(* IEC 61131-3 sources: B-R/Processes/EDT (part 4) *)

(* ---- EDTP4S1C_ACTION.st ---- *)
ACTION P4S1C_ACT:
	//设定时间
	FOR i := 0 TO EDTP4S1_STEP_NUM DO
		IF EDTP4S1C_ST[i] < T#5s THEN
			EDTP4S1C_ST[i] := T#5s;
		END_IF;
		EDTP4S1C_STEP[i].set_time := EDTP4S1C_ST[i];
	END_FOR;

	//流程步骤
	ProcessHandleFC(EDTP4S1C,EDTP4S1C_STEP[0],EDTP4S1_STEP_NUM);

	//object 手自动切换
	IF (EDTP4S1C.status.mode <> 0) AND (NOT EDTP4S1C.auto_mode_edge) THEN
		EDTP4S1C.auto_mode_edge := TRUE;
		EDTP4S1C.manual_mode_edge := FALSE;

		EDTXV1011.control.auto_operate := TRUE;
		EDTXV1022.control.auto_operate := TRUE;
		EDTP16.control.auto_operate := TRUE;
		EDTLV1002.control.auto_operate := TRUE;
		STFP06.control.auto_operate := TRUE;
		STFLV0602.control.auto_operate := TRUE;
		STFLV0601.control.auto_operate := TRUE;
		EDTLV1003.control.auto_operate := TRUE;
		EDTFQV1001C.control.auto_operate := TRUE;
		EDTTV1006B.control.auto_operate := TRUE;
		EDTXV1023.control.auto_operate := TRUE;
		EDTXV1018.control.auto_operate := TRUE;
		EDTTV1005A.control.auto_operate := TRUE;
		EDTTV1005B.control.auto_operate := TRUE;
		EDTTV1006A.control.auto_operate := TRUE;
		EDTXV1020.control.auto_operate := TRUE;
		EDTR04C.control.auto_operate := TRUE;
		EDTLV1004C.control.auto_operate := TRUE;
	END_IF;

	IF (EDTP4S1C.status.mode = 0) AND (NOT EDTP4S1C.manual_mode_edge) THEN
		EDTP4S1C.manual_mode_edge := TRUE;
		EDTP4S1C.auto_mode_edge := FALSE;

		EDTXV1011.control.manual_operate := TRUE;
		EDTXV1022.control.manual_operate := TRUE;
		EDTP16.control.manual_operate := TRUE;
		EDTLV1002.control.manual_operate := TRUE;
		STFP06.control.manual_operate := TRUE;
		STFLV0602.control.manual_operate := TRUE;
		STFLV0601.control.manual_operate := TRUE;
		EDTLV1003.control.manual_operate := TRUE;
		EDTFQV1001C.control.manual_operate := TRUE;
		EDTTV1006B.control.manual_operate := TRUE;
		EDTXV1023.control.manual_operate := TRUE;
		EDTXV1018.control.manual_operate := TRUE;
		EDTTV1005A.control.manual_operate := TRUE;
		EDTTV1005B.control.manual_operate := TRUE;
		EDTTV1006A.control.manual_operate := TRUE;
		EDTXV1020.control.manual_operate := TRUE;
		EDTR04C.control.manual_operate := TRUE;
		EDTLV1004C.control.manual_operate := TRUE;
	END_IF;

	//错误信号停机
	EDTP4S1C.input.error_signal := (EDTXV1011.status.valve_status >= 2) OR
	(EDTXV1022.status.valve_status >= 2) OR (EDTP16.status.motor_status >= 2) OR
	(EDTLV1002.status.valve_status >= 2) OR (STFP06.status.motor_status >= 2) OR (STFLV0602.status.valve_status >= 2) OR
	(STFLV0601.status.valve_status >= 2) OR (EDTLV1003.status.valve_status >= 2) OR (EDTFQV1001C.status.valve_status >= 2) OR
	(EDTTV1006B.status.valve_status >= 2) OR (EDTXV1023.status.valve_status >= 2) OR
	(EDTXV1018.status.valve_status >= 2) OR (EDTTV1005A.status.valve_status >= 2) OR (EDTTV1005B.status.valve_status >= 2) OR
	(EDTTV1006A.status.valve_status >= 2) OR (EDTR04C.status.motor_status >= 2) OR (EDTXV1020.status.valve_status >= 2);

	//EDTLV1004C自动补水
	//	IF EDTTIT1005.status.value >= EDTP4S1C_PARA_Temp7 THEN
	//		EDTLV1004C.input.auto_open_signal := TRUE;
	//	ELSIF EDTTIT1005.status.value <= (EDTP4S1C_PARA_Temp7 - EDTP4S1C_PARA_Temp8) THEN
	//		EDTLV1004C.input.auto_open_signal := FALSE;
	//	END_IF;
	IF r04c_water THEN
		CASE r04c_water_step OF
			0:
				EDTLV1004C.control.auto_operate := TRUE;
				r04c_water_step := 1;
			1:
				EDTLV1004C.input.auto_open_signal := TRUE;
				r04c_temp := EDTTIT1005.status.value;
				r04c_water_step := 2;
			2:
				IF r04c_temp - EDTTIT1005.status.value >= EDTP4S1C_PARA_Temp8 THEN
					EDTLV1004C.input.auto_open_signal := FALSE;
					r04c_water_step := 0;
					r04c_water := FALSE;
				END_IF;
		END_CASE;
	END_IF;

	IF EDTP4S1C.status.run_state = 1 THEN
		CASE EDTP4S1C.status.run_step OF
			0:
				IF NOT EDTP4S1C_STEP[0].done THEN
					EDTXV1011.control.auto_operate := TRUE;
					EDTXV1022.control.auto_operate := TRUE;
					EDTP16.control.auto_operate := TRUE;
					EDTLV1002.control.auto_operate := TRUE;
					STFP06.control.auto_operate := TRUE;
					STFLV0602.control.auto_operate := TRUE;
					STFLV0601.control.auto_operate := TRUE;
					EDTLV1003.control.auto_operate := TRUE;
					EDTFQV1001C.control.auto_operate := TRUE;
					EDTTV1006B.control.auto_operate := TRUE;
					EDTXV1023.control.auto_operate := TRUE;
					EDTXV1018.control.auto_operate := TRUE;
					EDTTV1005A.control.auto_operate := TRUE;
					EDTTV1005B.control.auto_operate := TRUE;
					EDTTV1006A.control.auto_operate := TRUE;
					EDTXV1020.control.auto_operate := TRUE;
					EDTR04C.control.auto_operate := TRUE;
					EDTLV1004C.control.auto_operate := TRUE;
					EDTP4S1C_STEP[0].done := TRUE;
				END_IF;
			1:
				//手动进DMSO和纯水
			2:
				EDTTV1005A.input.auto_open_signal := TRUE;
				EDTTV1005B.input.auto_open_signal := TRUE;
				EDTXV1023.input.auto_open_signal := TRUE;
				EDTXV1018.input.auto_open_signal := TRUE;
				EDTR04C.input.auto_run_signal := TRUE;
				EDTTV1006B.input.auto_open_signal := TRUE;
				EDTXV1020.input.auto_open_signal := TRUE;
				IF EDTXV1023.input.open_feedback_state AND EDTXV1018.input.open_feedback_state AND EDTR04C.input.run_feedback
					AND EDTTV1006B.input.open_feedback_state AND EDTXV1020.input.open_feedback_state THEN
					EDTP4S1C_STEP[2].done := TRUE;
				END_IF;
			3:
				CASE p4_step1_3c OF
					0:
						IF NOT EDTP4S1C_STEP[3].done THEN
							p4_step1_3c := 1;
						END_IF;
					1:
						R04C_heat := TRUE;
						p4_step1_3c := 2;
					2:
						IF EDTTIT1005.status.value >= EDTP4S1C_PARA_Temp1 THEN
							EDTTV1006B.input.auto_open_signal := FALSE;
							IF EDTTV1006B.input.close_feedback_state THEN
								EDTTV1006A.input.auto_open_signal := TRUE;
								IF EDTTV1006A.input.open_feedback_state THEN
									p4_step1_3c := 3;
								END_IF;
							END_IF;
						END_IF;
					3:
						TON_77.PT := DINT_TO_TIME(EDTP4S1C_PARA_T4 * 3600 * 1000);
						IF EDTTIT1005.status.value >= EDTP4S1C_PARA_Temp2 THEN
							R04C_heat := FALSE;
							R04C_hold := TRUE;
							TON_77.IN := TRUE;
						END_IF;
						IF TON_77.Q THEN
							TON_77.IN := FALSE;
							p4_step1_3c := 4;
						END_IF;
					4:
						p4_step1_3c := 0;
						EDTP4S1C_STEP[3].done := TRUE;
				END_CASE;
				TON_77();
			4:
				//人工取样,确认反应结束
			5:
				R04C_hold := FALSE;
				EDTTV1005A.input.auto_open_signal := FALSE;
				EDTTV1005B.input.auto_open_signal := FALSE;
				IF EDTTV1005A.input.close_feedback_state AND EDTTV1005B.input.close_feedback_state THEN
					EDTP4S1C_STEP[5].done := TRUE;
				END_IF;
			6:
				IF EDTTIT1005.status.value <= EDTP4S1C_PARA_Temp5 THEN
					//					EDTXV1023.input.auto_open_signal := FALSE;
					//					EDTXV1018.input.auto_open_signal := FALSE;
					EDTTV1006A.input.auto_open_signal := FALSE;
				END_IF;
				IF (*EDTXV1023.input.close_feedback_state AND EDTXV1018.input.close_feedback_state AND *)(NOT EDTR04C.input.run_feedback)
					AND EDTTV1006A.input.close_feedback_state THEN
					EDTP4S1C_STEP[6].done := TRUE;
				END_IF;
			7:
				//转移
			8:
				EDTR04C.input.auto_run_signal := FALSE;
				IF NOT EDTR04C.input.run_feedback THEN
					EDTP4S1C_STEP[8].done := TRUE;
				END_IF;
		END_CASE;
	END_IF;

	Slope_2(value := EDTTIT1005.status.value, sample_time := EDTP4S1C_PARA_T5);

	IF R04C_heat THEN
		IF Slope_2.out <= EDTP4S1C_PARA_Slope1 THEN
			EDTTV1005A.input.auto_open_signal := TRUE;
			EDTTV1005B.input.auto_open_signal := TRUE;
		END_IF;
		IF Slope_2.out > EDTP4S1C_PARA_Slope1 AND Slope_2.out <= EDTP4S1C_PARA_Slope2 THEN
			EDTTV1005A.input.auto_open_signal := TRUE;
			EDTTV1005B.input.auto_open_signal := FALSE;
		END_IF;
		IF Slope_2.out > EDTP4S1C_PARA_Slope2 AND Slope_2.out <= EDTP4S1C_PARA_Slope3 THEN
			EDTTV1005A.input.auto_open_signal := FALSE;
			EDTTV1005B.input.auto_open_signal := TRUE;
		END_IF;
		IF Slope_2.out > EDTP4S1C_PARA_Slope3 THEN
			EDTTV1005A.input.auto_open_signal := FALSE;
			EDTTV1005B.input.auto_open_signal := FALSE;
		END_IF;
	END_IF;

	//155-158 大  158-162小阀 162都关
	IF R04C_hold THEN
		IF EDTTIT1005.status.value < EDTP4S1C_PARA_Temp2 THEN
			EDTTV1005A.input.auto_open_signal := TRUE;
			EDTTV1005B.input.auto_open_signal := TRUE;
		END_IF;
		IF EDTTIT1005.status.value < EDTP4S1C_PARA_Temp3 AND EDTTIT1005.status.value >= (EDTP4S1C_PARA_Temp2 + EDTP4S1C_PARA_Temp6) THEN
			EDTTV1005A.input.auto_open_signal := TRUE;
			EDTTV1005B.input.auto_open_signal := FALSE;
		END_IF;
		IF EDTTIT1005.status.value < EDTP4S1C_PARA_Temp4 AND EDTTIT1005.status.value >= (EDTP4S1C_PARA_Temp3 + EDTP4S1C_PARA_Temp6) THEN
			EDTTV1005A.input.auto_open_signal := FALSE;
			EDTTV1005B.input.auto_open_signal := TRUE;
		END_IF;
		IF EDTTIT1005.status.value >= (EDTP4S1C_PARA_Temp4 + EDTP4S1C_PARA_Temp6) THEN
			EDTTV1005A.input.auto_open_signal := FALSE;
			EDTTV1005B.input.auto_open_signal := FALSE;
		END_IF;
	END_IF;

	//======================================================================================================
	//DMSO进料
	//从罐区进料
	IF pot_to_r04_c THEN
		CASE pot_to_r04_c_step OF
			0:
				EDTFQV1001C.input.auto_open_signal := TRUE;
				EDTLV1003.input.auto_open_signal := TRUE;
				STFLV0601.input.auto_open_signal := FALSE;
				STFLV0602.input.auto_open_signal := FALSE;
				IF EDTFQV1001C.input.open_feedback_state AND EDTLV1003.input.open_feedback_state AND
					STFLV0601.input.close_feedback_state AND STFLV0602.input.close_feedback_state THEN
					pot_to_r04_c_step := 1;
				END_IF;
			1:
				LiquidTransfer_30(sp_time := DINT_TO_TIME(EDTP4S1C_PARA_T2 * 1000),
				sp_accumulation := EDTP4S1C_PARA_AC1,
				done := pot_to_r04_c_step_1_done,
				flowmeter := EDTFQIT1001);
				STFP06.input.auto_run_signal := LiquidTransfer_30.run;
				IF pot_to_r04_c_step_1_done AND (NOT STFP06.input.run_feedback) AND (NOT STFP06.input.auto_run_signal) THEN
					pot_to_r04_c_step_1_done := FALSE;
					pot_to_r04_c_step := 2;
				END_IF;
			2:
				IF EDTFQIT1001.flowrate <= flowrate_threshold THEN
					pot_to_r04_c_step := 3;
				END_IF;
			3:
				EDTFQV1001C.input.auto_open_signal := FALSE;
				EDTLV1003.input.auto_open_signal := FALSE;
				IF EDTFQV1001C.input.close_feedback_state AND EDTLV1003.input.close_feedback_state THEN
					pot_to_r04_c_step := 0;
					pot_to_r04_c := FALSE;
				END_IF;
		END_CASE;
	END_IF;

	//从V52进料
	IF v52_to_r04_c THEN
		CASE v52_to_r04_c_step OF
			0:
				EDTFQV1001C.input.auto_open_signal := TRUE;
				EDTLV1002.input.auto_open_signal := TRUE;
				IF EDTFQV1001C.input.open_feedback_state AND EDTLV1002.input.open_feedback_state THEN
					v52_to_r04_c_step := 1;
				END_IF;
			1:
				LiquidTransfer_31(sp_time := DINT_TO_TIME(EDTP4S1C_PARA_T3 * 1000),
				sp_accumulation := EDTP4S1C_PARA_AC2,
				done := v52_to_r04_c_step_1_done,
				flowmeter := EDTFQIT1001);
				EDTP16.input.auto_run_signal := LiquidTransfer_31.run;
				IF v52_to_r04_c_step_1_done AND (NOT EDTP16.input.run_feedback) AND (NOT EDTP16.input.auto_run_signal) THEN
					v52_to_r04_c_step_1_done := FALSE;
					v52_to_r04_c_step := 2;
				END_IF;
			2:
				IF EDTFQIT1001.flowrate <= flowrate_threshold THEN
					v52_to_r04_c_step := 3;
				END_IF;
			3:
				EDTFQV1001C.input.auto_open_signal := FALSE;
				EDTLV1002.input.auto_open_signal := FALSE;
				IF EDTFQV1001C.input.close_feedback_state AND EDTLV1002.input.close_feedback_state THEN
					v52_to_r04_c_step := 0;
					v52_to_r04_c := FALSE;
				END_IF;
		END_CASE;
	END_IF;

	//=======================================================================================================
	//人工确认步骤可用
	IF (EDTP4S1C.status.run_state) AND (NOT EDTP4S1C_STEP[EDTP4S1C.status.run_step].done AND ((EDTP4S1C.status.run_step = 1) OR (EDTP4S1C.status.run_step = 4) OR (EDTP4S1C.status.run_step = 7))) THEN
		EDTP4S1C.status.confirm_enable := TRUE;
	ELSE
		EDTP4S1C.status.confirm_enable := FALSE;
	END_IF;
END_ACTION

(* ---- EDTP4S1D_ACTION.st ---- *)
ACTION P4S1D_ACT:
	//设定时间
	FOR i := 0 TO EDTP4S1_STEP_NUM DO
		IF EDTP4S1D_ST[i] < T#5s THEN
			EDTP4S1D_ST[i] := T#5s;
		END_IF;
		EDTP4S1D_STEP[i].set_time := EDTP4S1D_ST[i];
	END_FOR;

	//流程步骤
	ProcessHandleFC(EDTP4S1D,EDTP4S1D_STEP[0],EDTP4S1_STEP_NUM);

	//object 手自动切换
	IF (EDTP4S1D.status.mode <> 0) AND (NOT EDTP4S1D.auto_mode_edge) THEN
		EDTP4S1D.auto_mode_edge := TRUE;
		EDTP4S1D.manual_mode_edge := FALSE;

		EDTXV1011.control.auto_operate := TRUE;
		EDTXV1022.control.auto_operate := TRUE;
		EDTP16.control.auto_operate := TRUE;
		EDTLV1002.control.auto_operate := TRUE;
		STFP06.control.auto_operate := TRUE;
		STFLV0602.control.auto_operate := TRUE;
		STFLV0601.control.auto_operate := TRUE;
		EDTLV1003.control.auto_operate := TRUE;
		EDTFQV1001D.control.auto_operate := TRUE;
		EDTTV1008B.control.auto_operate := TRUE;
		EDTXV1024.control.auto_operate := TRUE;
		EDTXV1019.control.auto_operate := TRUE;
		EDTTV1007A.control.auto_operate := TRUE;
		EDTTV1007B.control.auto_operate := TRUE;
		EDTTV1008A.control.auto_operate := TRUE;
		EDTXV1021.control.auto_operate := TRUE;
		EDTR04D.control.auto_operate := TRUE;
		EDTLV1004D.control.auto_operate := TRUE;
	END_IF;

	IF (EDTP4S1D.status.mode = 0) AND (NOT EDTP4S1D.manual_mode_edge) THEN
		EDTP4S1D.manual_mode_edge := TRUE;
		EDTP4S1D.auto_mode_edge := FALSE;

		EDTXV1011.control.manual_operate := TRUE;
		EDTXV1022.control.manual_operate := TRUE;
		EDTP16.control.manual_operate := TRUE;
		EDTLV1002.control.manual_operate := TRUE;
		STFP06.control.manual_operate := TRUE;
		STFLV0602.control.manual_operate := TRUE;
		STFLV0601.control.manual_operate := TRUE;
		EDTLV1003.control.manual_operate := TRUE;
		EDTFQV1001D.control.manual_operate := TRUE;
		EDTTV1008B.control.manual_operate := TRUE;
		EDTXV1024.control.manual_operate := TRUE;
		EDTXV1019.control.manual_operate := TRUE;
		EDTTV1007A.control.manual_operate := TRUE;
		EDTTV1007B.control.manual_operate := TRUE;
		EDTTV1008A.control.manual_operate := TRUE;
		EDTXV1021.control.manual_operate := TRUE;
		EDTR04D.control.manual_operate := TRUE;
		EDTLV1004D.control.manual_operate := TRUE;
	END_IF;

	//错误信号停机
	EDTP4S1D.input.error_signal := (EDTXV1011.status.valve_status >= 2) OR
	(EDTXV1022.status.valve_status >= 2) OR (EDTP16.status.motor_status >= 2) OR
	(EDTLV1002.status.valve_status >= 2) OR (STFP06.status.motor_status >= 2) OR (STFLV0602.status.valve_status >= 2) OR
	(STFLV0601.status.valve_status >= 2) OR (EDTLV1003.status.valve_status >= 2) OR (EDTFQV1001D.status.valve_status >= 2) OR
	(EDTTV1008B.status.valve_status >= 2) OR (EDTXV1024.status.valve_status >= 2) OR
	(EDTXV1019.status.valve_status >= 2) OR (EDTTV1007A.status.valve_status >= 2) OR (EDTTV1007B.status.valve_status >= 2) OR
	(EDTTV1008A.status.valve_status >= 2) OR (EDTR04D.status.motor_status >= 2) OR (EDTXV1021.status.valve_status >= 2);

	//EDTLV1004D自动补水
	//	IF EDTTIT1007.status.value >= EDTP4S1D_PARA_Temp7 THEN
	//		EDTLV1004D.input.auto_open_signal := TRUE;
	//	ELSIF EDTTIT1007.status.value <= (EDTP4S1D_PARA_Temp7 - EDTP4S1D_PARA_Temp8) THEN
	//		EDTLV1004D.input.auto_open_signal := FALSE;
	//	END_IF;
	IF r04d_water THEN
		CASE r04d_water_step OF
			0:
				EDTLV1004D.control.auto_operate := TRUE;
				r04d_water_step := 1;
			1:
				EDTLV1004D.input.auto_open_signal := TRUE;
				r04d_temp := EDTTIT1007.status.value;
				r04d_water_step := 2;
			2:
				IF r04d_temp - EDTTIT1007.status.value >= EDTP4S1D_PARA_Temp8 THEN
					EDTLV1004D.input.auto_open_signal := FALSE;
					r04d_water_step := 0;
					r04d_water := FALSE;
				END_IF;
		END_CASE;
	END_IF;

	IF EDTP4S1D.status.run_state = 1 THEN
		CASE EDTP4S1D.status.run_step OF
			0:
				IF NOT EDTP4S1D_STEP[0].done THEN
					EDTXV1011.control.auto_operate := TRUE;
					EDTXV1022.control.auto_operate := TRUE;
					EDTP16.control.auto_operate := TRUE;
					EDTLV1002.control.auto_operate := TRUE;
					STFP06.control.auto_operate := TRUE;
					STFLV0602.control.auto_operate := TRUE;
					STFLV0601.control.auto_operate := TRUE;
					EDTLV1003.control.auto_operate := TRUE;
					EDTFQV1001D.control.auto_operate := TRUE;
					EDTTV1008B.control.auto_operate := TRUE;
					EDTXV1024.control.auto_operate := TRUE;
					EDTXV1019.control.auto_operate := TRUE;
					EDTTV1007A.control.auto_operate := TRUE;
					EDTTV1007B.control.auto_operate := TRUE;
					EDTTV1008A.control.auto_operate := TRUE;
					EDTXV1021.control.auto_operate := TRUE;
					EDTR04D.control.auto_operate := TRUE;
					EDTLV1004D.control.auto_operate := TRUE;
					EDTP4S1D_STEP[0].done := TRUE;
				END_IF;
			1:
				//手动进DMSO和纯水
			2:
				EDTTV1007A.input.auto_open_signal := TRUE;
				EDTTV1007B.input.auto_open_signal := TRUE;
				EDTXV1024.input.auto_open_signal := TRUE;
				EDTXV1019.input.auto_open_signal := TRUE;
				EDTR04D.input.auto_run_signal := TRUE;
				EDTTV1008B.input.auto_open_signal := TRUE;
				EDTXV1021.input.auto_open_signal := TRUE;
				IF EDTXV1024.input.open_feedback_state AND EDTXV1019.input.open_feedback_state AND EDTR04D.input.run_feedback
					AND EDTTV1008B.input.open_feedback_state AND EDTXV1021.input.open_feedback_state THEN
					EDTP4S1D_STEP[2].done := TRUE;
				END_IF;
			3:
				CASE p4_step1_3d OF
					0:
						IF NOT EDTP4S1D_STEP[3].done THEN
							p4_step1_3d := 1;
						END_IF;
					1:
						R04D_heat := TRUE;
						p4_step1_3d := 2;
					2:
						IF EDTTIT1007.status.value >= EDTP4S1D_PARA_Temp1 THEN
							EDTTV1008B.input.auto_open_signal := FALSE;
							IF EDTTV1008B.input.close_feedback_state THEN
								EDTTV1008A.input.auto_open_signal := TRUE;
								IF EDTTV1008A.input.open_feedback_state THEN
									p4_step1_3d := 3;
								END_IF;
							END_IF;
						END_IF;
					3:
						TON_79.PT := DINT_TO_TIME(EDTP4S1D_PARA_T4 * 3600 * 1000);
						IF EDTTIT1007.status.value >= EDTP4S1D_PARA_Temp2 THEN
							R04D_heat := FALSE;
							R04D_hold := TRUE;
							TON_79.IN := TRUE;
						END_IF;
						IF TON_79.Q THEN
							TON_79.IN := FALSE;
							p4_step1_3d := 4;
						END_IF;
					4:
						p4_step1_3d := 0;
						EDTP4S1D_STEP[3].done := TRUE;
				END_CASE;
				TON_79();
			4:
				//人工取样,确认反应结束
			5:
				R04D_hold := FALSE;
				EDTTV1007A.input.auto_open_signal := FALSE;
				EDTTV1007B.input.auto_open_signal := FALSE;
				IF EDTTV1007A.input.close_feedback_state AND EDTTV1007B.input.close_feedback_state THEN
					EDTP4S1D_STEP[5].done := TRUE;
				END_IF;
			6:
				IF EDTTIT1007.status.value <= EDTP4S1D_PARA_Temp5 THEN
					//					EDTXV1024.input.auto_open_signal := FALSE;
					//					EDTXV1019.input.auto_open_signal := FALSE;
					EDTTV1008A.input.auto_open_signal := FALSE;
				END_IF;
				IF (*EDTXV1024.input.close_feedback_state AND EDTXV1019.input.close_feedback_state AND *)(NOT EDTR04D.input.run_feedback)
					AND EDTTV1008A.input.close_feedback_state THEN
					EDTP4S1D_STEP[6].done := TRUE;
				END_IF;
			7:
				//转移
			8:
				EDTR04D.input.auto_run_signal := FALSE;
				IF NOT EDTR04D.input.run_feedback THEN
					EDTP4S1D_STEP[8].done := TRUE;
				END_IF;
		END_CASE;
	END_IF;

	Slope_3(value := EDTTIT1007.status.value, sample_time := EDTP4S1D_PARA_T5);

	IF R04D_heat THEN
		IF Slope_3.out <= EDTP4S1D_PARA_Slope1 THEN
			EDTTV1007A.input.auto_open_signal := TRUE;
			EDTTV1007B.input.auto_open_signal := TRUE;
		END_IF;
		IF Slope_3.out > EDTP4S1D_PARA_Slope1 AND Slope_3.out <= EDTP4S1D_PARA_Slope2 THEN
			EDTTV1007A.input.auto_open_signal := TRUE;
			EDTTV1007B.input.auto_open_signal := FALSE;
		END_IF;
		IF Slope_3.out > EDTP4S1D_PARA_Slope2 AND Slope_3.out <= EDTP4S1D_PARA_Slope3 THEN
			EDTTV1007A.input.auto_open_signal := FALSE;
			EDTTV1007B.input.auto_open_signal := TRUE;
		END_IF;
		IF Slope_3.out > EDTP4S1D_PARA_Slope3 THEN
			EDTTV1007A.input.auto_open_signal := FALSE;
			EDTTV1007B.input.auto_open_signal := FALSE;
		END_IF;
	END_IF;

	//155-158 大  158-162小阀 162都关
	IF R04D_hold THEN
		IF EDTTIT1007.status.value < EDTP4S1D_PARA_Temp2 THEN
			EDTTV1007A.input.auto_open_signal := TRUE;
			EDTTV1007B.input.auto_open_signal := TRUE;
		END_IF;
		IF EDTTIT1007.status.value < EDTP4S1D_PARA_Temp3 AND EDTTIT1007.status.value >= (EDTP4S1D_PARA_Temp2 + EDTP4S1D_PARA_Temp6) THEN
			EDTTV1007A.input.auto_open_signal := TRUE;
			EDTTV1007B.input.auto_open_signal := FALSE;
		END_IF;
		IF EDTTIT1007.status.value < EDTP4S1D_PARA_Temp4 AND EDTTIT1007.status.value >= (EDTP4S1D_PARA_Temp3 + EDTP4S1D_PARA_Temp6) THEN
			EDTTV1007A.input.auto_open_signal := FALSE;
			EDTTV1007B.input.auto_open_signal := TRUE;
		END_IF;
		IF EDTTIT1007.status.value >= (EDTP4S1D_PARA_Temp4 + EDTP4S1D_PARA_Temp6) THEN
			EDTTV1007A.input.auto_open_signal := FALSE;
			EDTTV1007B.input.auto_open_signal := FALSE;
		END_IF;
	END_IF;

	//======================================================================================================
	//DMSO进料
	//从罐区进料
	IF pot_to_r04_d THEN
		CASE pot_to_r04_d_step OF
			0:
				EDTFQV1001D.input.auto_open_signal := TRUE;
				EDTLV1003.input.auto_open_signal := TRUE;
				STFLV0601.input.auto_open_signal := FALSE;
				STFLV0602.input.auto_open_signal := FALSE;
				IF EDTFQV1001D.input.open_feedback_state AND EDTLV1003.input.open_feedback_state AND
					STFLV0601.input.close_feedback_state AND STFLV0602.input.close_feedback_state THEN
					pot_to_r04_d_step := 1;
				END_IF;
			1:
				LiquidTransfer_32(sp_time := DINT_TO_TIME(EDTP4S1D_PARA_T2 * 1000),
				sp_accumulation := EDTP4S1D_PARA_AC1,
				done := pot_to_r04_d_step_1_done,
				flowmeter := EDTFQIT1001);
				STFP06.input.auto_run_signal := LiquidTransfer_32.run;
				IF pot_to_r04_d_step_1_done AND (NOT STFP06.input.run_feedback) AND (NOT STFP06.input.auto_run_signal) THEN
					pot_to_r04_d_step_1_done := FALSE;
					pot_to_r04_d_step := 2;
				END_IF;
			2:
				IF EDTFQIT1001.flowrate <= flowrate_threshold THEN
					pot_to_r04_d_step := 3;
				END_IF;
			3:
				EDTFQV1001D.input.auto_open_signal := FALSE;
				EDTLV1003.input.auto_open_signal := FALSE;
				IF EDTFQV1001D.input.close_feedback_state AND EDTLV1003.input.close_feedback_state THEN
					pot_to_r04_d_step := 0;
					pot_to_r04_d := FALSE;
				END_IF;
		END_CASE;
	END_IF;

	//从V52进料
	IF v52_to_r04_d THEN
		CASE v52_to_r04_d_step OF
			0:
				EDTFQV1001D.input.auto_open_signal := TRUE;
				EDTLV1002.input.auto_open_signal := TRUE;
				IF EDTFQV1001D.input.open_feedback_state AND EDTLV1002.input.open_feedback_state THEN
					v52_to_r04_d_step := 1;
				END_IF;
			1:
				LiquidTransfer_33(sp_time := DINT_TO_TIME(EDTP4S1D_PARA_T3 * 1000),
				sp_accumulation := EDTP4S1D_PARA_AC2,
				done := v52_to_r04_d_step_1_done,
				flowmeter := EDTFQIT1001);
				EDTP16.input.auto_run_signal := LiquidTransfer_33.run;
				IF v52_to_r04_d_step_1_done AND (NOT EDTP16.input.run_feedback) AND (NOT EDTP16.input.auto_run_signal) THEN
					v52_to_r04_d_step_1_done := FALSE;
					v52_to_r04_d_step := 2;
				END_IF;
			2:
				IF EDTFQIT1001.flowrate <= flowrate_threshold THEN
					v52_to_r04_d_step := 3;
				END_IF;
			3:
				EDTFQV1001D.input.auto_open_signal := FALSE;
				EDTLV1002.input.auto_open_signal := FALSE;
				IF EDTFQV1001D.input.close_feedback_state AND EDTLV1002.input.close_feedback_state THEN
					v52_to_r04_d_step := 0;
					v52_to_r04_d := FALSE;
				END_IF;
		END_CASE;
	END_IF;

	//=======================================================================================================
	//人工确认步骤可用
	IF (EDTP4S1D.status.run_state) AND (NOT EDTP4S1D_STEP[EDTP4S1D.status.run_step].done AND ((EDTP4S1D.status.run_step = 1) OR (EDTP4S1D.status.run_step = 4) OR (EDTP4S1D.status.run_step = 7))) THEN
		EDTP4S1D.status.confirm_enable := TRUE;
	ELSE
		EDTP4S1D.status.confirm_enable := FALSE;
	END_IF;
END_ACTION

(* ---- EDTP4S1E_ACTION.st ---- *)
ACTION P4S1E_ACT:
	//设定时间
	FOR i := 0 TO EDTP4S1_STEP_NUM DO
		IF EDTP4S1E_ST[i] < T#5s THEN
			EDTP4S1E_ST[i] := T#5s;
		END_IF;
		EDTP4S1E_STEP[i].set_time := EDTP4S1E_ST[i];
	END_FOR;

	//流程步骤
	ProcessHandleFC(EDTP4S1E,EDTP4S1E_STEP[0],EDTP4S1_STEP_NUM);

	//object 手自动切换
	IF (EDTP4S1E.status.mode <> 0) AND (NOT EDTP4S1E.auto_mode_edge) THEN
		EDTP4S1E.auto_mode_edge := TRUE;
		EDTP4S1E.manual_mode_edge := FALSE;

		EDTXV1011.control.auto_operate := TRUE;
		EDTXV1031.control.auto_operate := TRUE;
		EDTP16.control.auto_operate := TRUE;
		EDTLV1002.control.auto_operate := TRUE;
		STFP06.control.auto_operate := TRUE;
		STFLV0602.control.auto_operate := TRUE;
		STFLV0601.control.auto_operate := TRUE;
		EDTLV1003.control.auto_operate := TRUE;
		EDTFQV1001E.control.auto_operate := TRUE;
		EDTTV1010B.control.auto_operate := TRUE;
		EDTXV1032.control.auto_operate := TRUE;
		EDTXV1027.control.auto_operate := TRUE;
		EDTTV1009A.control.auto_operate := TRUE;
		EDTTV1009B.control.auto_operate := TRUE;
		EDTTV1010A.control.auto_operate := TRUE;
		EDTXV1029.control.auto_operate := TRUE;
		EDTR04E.control.auto_operate := TRUE;
		EDTLV1004E.control.auto_operate := TRUE;
	END_IF;

	IF (EDTP4S1E.status.mode = 0) AND (NOT EDTP4S1E.manual_mode_edge) THEN
		EDTP4S1E.manual_mode_edge := TRUE;
		EDTP4S1E.auto_mode_edge := FALSE;

		EDTXV1011.control.manual_operate := TRUE;
		EDTXV1031.control.manual_operate := TRUE;
		EDTP16.control.manual_operate := TRUE;
		EDTLV1002.control.manual_operate := TRUE;
		STFP06.control.manual_operate := TRUE;
		STFLV0602.control.manual_operate := TRUE;
		STFLV0601.control.manual_operate := TRUE;
		EDTLV1003.control.manual_operate := TRUE;
		EDTFQV1001E.control.manual_operate := TRUE;
		EDTTV1010B.control.manual_operate := TRUE;
		EDTXV1032.control.manual_operate := TRUE;
		EDTXV1027.control.manual_operate := TRUE;
		EDTTV1009A.control.manual_operate := TRUE;
		EDTTV1009B.control.manual_operate := TRUE;
		EDTTV1010A.control.manual_operate := TRUE;
		EDTXV1029.control.manual_operate := TRUE;
		EDTR04E.control.manual_operate := TRUE;
		EDTLV1004E.control.manual_operate := TRUE;
	END_IF;

	//错误信号停机
	EDTP4S1E.input.error_signal := (EDTXV1011.status.valve_status >= 2) OR
	(EDTXV1031.status.valve_status >= 2) OR (EDTP16.status.motor_status >= 2) OR
	(EDTLV1002.status.valve_status >= 2) OR (STFP06.status.motor_status >= 2) OR (STFLV0602.status.valve_status >= 2) OR
	(STFLV0601.status.valve_status >= 2) OR (EDTLV1003.status.valve_status >= 2) OR (EDTFQV1001E.status.valve_status >= 2) OR
	(EDTTV1010B.status.valve_status >= 2) OR (EDTXV1032.status.valve_status >= 2) OR
	(EDTXV1027.status.valve_status >= 2) OR (EDTTV1009A.status.valve_status >= 2) OR (EDTTV1009B.status.valve_status >= 2) OR
	(EDTTV1010A.status.valve_status >= 2) OR (EDTR04E.status.motor_status >= 2) OR (EDTXV1029.status.valve_status >= 2);

	//EDTLV1004E自动补水
	//	IF EDTTIT1009.status.value >= EDTP4S1E_PARA_Temp7 THEN
	//		EDTLV1004E.input.auto_open_signal := TRUE;
	//	ELSIF EDTTIT1009.status.value <= (EDTP4S1E_PARA_Temp7 - EDTP4S1E_PARA_Temp8) THEN
	//		EDTLV1004E.input.auto_open_signal := FALSE;
	//	END_IF;
	IF r04e_water THEN
		CASE r04e_water_step OF
			0:
				EDTLV1004E.control.auto_operate := TRUE;
				r04e_water_step := 1;
			1:
				EDTLV1004E.input.auto_open_signal := TRUE;
				r04e_temp := EDTTIT1009.status.value;
				r04e_water_step := 2;
			2:
				IF r04e_temp - EDTTIT1009.status.value >= EDTP4S1E_PARA_Temp8 THEN
					EDTLV1004E.input.auto_open_signal := FALSE;
					r04e_water_step := 0;
					r04e_water := FALSE;
				END_IF;
		END_CASE;
	END_IF;

	IF EDTP4S1E.status.run_state = 1 THEN
		CASE EDTP4S1E.status.run_step OF
			0:
				IF NOT EDTP4S1E_STEP[0].done THEN
					EDTXV1011.control.auto_operate := TRUE;
					EDTXV1031.control.auto_operate := TRUE;
					EDTP16.control.auto_operate := TRUE;
					EDTLV1002.control.auto_operate := TRUE;
					STFP06.control.auto_operate := TRUE;
					STFLV0602.control.auto_operate := TRUE;
					STFLV0601.control.auto_operate := TRUE;
					EDTLV1003.control.auto_operate := TRUE;
					EDTFQV1001E.control.auto_operate := TRUE;
					EDTTV1010B.control.auto_operate := TRUE;
					EDTXV1032.control.auto_operate := TRUE;
					EDTXV1027.control.auto_operate := TRUE;
					EDTTV1009A.control.auto_operate := TRUE;
					EDTTV1009B.control.auto_operate := TRUE;
					EDTTV1010A.control.auto_operate := TRUE;
					EDTXV1029.control.auto_operate := TRUE;
					EDTR04E.control.auto_operate := TRUE;
					EDTLV1004E.control.auto_operate := TRUE;
					EDTP4S1E_STEP[0].done := TRUE;
				END_IF;
			1:
				//手动进DMSO和纯水
			2:
				EDTTV1009A.input.auto_open_signal := TRUE;
				EDTTV1009B.input.auto_open_signal := TRUE;
				EDTXV1032.input.auto_open_signal := TRUE;
				EDTXV1027.input.auto_open_signal := TRUE;
				EDTR04E.input.auto_run_signal := TRUE;
				EDTTV1010B.input.auto_open_signal := TRUE;
				EDTXV1029.input.auto_open_signal := TRUE;
				IF EDTXV1032.input.open_feedback_state AND EDTXV1027.input.open_feedback_state AND EDTR04E.input.run_feedback
					AND EDTTV1010B.input.open_feedback_state AND EDTXV1029.input.open_feedback_state THEN
					EDTP4S1E_STEP[2].done := TRUE;
				END_IF;
			3:
				CASE p4_step1_3e OF
					0:
						IF NOT EDTP4S1E_STEP[3].done THEN
							p4_step1_3e := 1;
						END_IF;
					1:
						R04E_heat := TRUE;
						p4_step1_3e := 2;
					2:
						IF EDTTIT1009.status.value >= EDTP4S1E_PARA_Temp1 THEN
							EDTTV1010B.input.auto_open_signal := FALSE;
							IF EDTTV1010B.input.close_feedback_state THEN
								EDTTV1010A.input.auto_open_signal := TRUE;
								IF EDTTV1010A.input.open_feedback_state THEN
									p4_step1_3e := 3;
								END_IF;
							END_IF;
						END_IF;

					3:
						TON_80.PT := DINT_TO_TIME(EDTP4S1E_PARA_T4 * 3600 * 1000);
						IF EDTTIT1009.status.value >= EDTP4S1E_PARA_Temp2 THEN
							R04E_heat := FALSE;
							R04E_hold := TRUE;
							TON_80.IN := TRUE;
						END_IF;
						IF TON_80.Q THEN
							TON_80.IN := FALSE;
							p4_step1_3e := 4;
						END_IF;
					4:
						p4_step1_3e := 0;
						EDTP4S1E_STEP[3].done := TRUE;
				END_CASE;
				TON_80();
			4:
				//人工取样,确认反应结束
			5:
				R04E_hold := FALSE;
				EDTTV1009A.input.auto_open_signal := FALSE;
				EDTTV1009B.input.auto_open_signal := FALSE;
				IF EDTTV1009A.input.close_feedback_state AND EDTTV1009B.input.close_feedback_state THEN
					EDTP4S1E_STEP[5].done := TRUE;
				END_IF;
			6:
				IF EDTTIT1009.status.value <= EDTP4S1E_PARA_Temp5 THEN
					//					EDTXV1032.input.auto_open_signal := FALSE;
					//					EDTXV1027.input.auto_open_signal := FALSE;
					EDTTV1010A.input.auto_open_signal := FALSE;
				END_IF;
				IF (*EDTXV1032.input.close_feedback_state AND EDTXV1027.input.close_feedback_state AND *)(NOT EDTR04E.input.run_feedback)
					AND EDTTV1010A.input.close_feedback_state THEN
					EDTP4S1E_STEP[6].done := TRUE;
				END_IF;
			7:
				//转移
			8:
				EDTR04E.input.auto_run_signal := FALSE;
				IF NOT EDTR04E.input.run_feedback THEN
					EDTP4S1E_STEP[8].done := TRUE;
				END_IF;
		END_CASE;
	END_IF;

	Slope_4(value := EDTTIT1009.status.value, sample_time := EDTP4S1E_PARA_T5);

	IF R04E_heat THEN
		IF Slope_4.out <= EDTP4S1E_PARA_Slope1 THEN
			EDTTV1009A.input.auto_open_signal := TRUE;
			EDTTV1009B.input.auto_open_signal := TRUE;
		END_IF;
		IF Slope_4.out > EDTP4S1E_PARA_Slope1 AND Slope_4.out <= EDTP4S1E_PARA_Slope2 THEN
			EDTTV1009A.input.auto_open_signal := TRUE;
			EDTTV1009B.input.auto_open_signal := FALSE;
		END_IF;
		IF Slope_4.out > EDTP4S1E_PARA_Slope2 AND Slope_4.out <= EDTP4S1E_PARA_Slope3 THEN
			EDTTV1009A.input.auto_open_signal := FALSE;
			EDTTV1009B.input.auto_open_signal := TRUE;
		END_IF;
		IF Slope_4.out > EDTP4S1E_PARA_Slope3 THEN
			EDTTV1009A.input.auto_open_signal := FALSE;
			EDTTV1009B.input.auto_open_signal := FALSE;
		END_IF;
	END_IF;

	//155-158 大  158-162小阀 162都关
	IF R04E_hold THEN
		IF EDTTIT1009.status.value < EDTP4S1E_PARA_Temp2 THEN
			EDTTV1009A.input.auto_open_signal := TRUE;
			EDTTV1009B.input.auto_open_signal := TRUE;
		END_IF;
		IF EDTTIT1009.status.value < EDTP4S1E_PARA_Temp3 AND EDTTIT1009.status.value >= (EDTP4S1E_PARA_Temp2 + EDTP4S1E_PARA_Temp6) THEN
			EDTTV1009A.input.auto_open_signal := TRUE;
			EDTTV1009B.input.auto_open_signal := FALSE;
		END_IF;
		IF EDTTIT1009.status.value < EDTP4S1E_PARA_Temp4 AND EDTTIT1009.status.value >= (EDTP4S1E_PARA_Temp3 + EDTP4S1E_PARA_Temp6) THEN
			EDTTV1009A.input.auto_open_signal := FALSE;
			EDTTV1009B.input.auto_open_signal := TRUE;
		END_IF;
		IF EDTTIT1009.status.value >= (EDTP4S1E_PARA_Temp4 + EDTP4S1E_PARA_Temp6) THEN
			EDTTV1009A.input.auto_open_signal := FALSE;
			EDTTV1009B.input.auto_open_signal := FALSE;
		END_IF;
	END_IF;

	//======================================================================================================
	//DMSO进料
	//从罐区进料
	IF pot_to_r04_e THEN
		CASE pot_to_r04_e_step OF
			0:
				EDTFQV1001E.input.auto_open_signal := TRUE;
				EDTLV1003.input.auto_open_signal := TRUE;
				STFLV0601.input.auto_open_signal := FALSE;
				STFLV0602.input.auto_open_signal := FALSE;
				IF EDTFQV1001E.input.open_feedback_state AND EDTLV1003.input.open_feedback_state AND
					STFLV0601.input.close_feedback_state AND STFLV0602.input.close_feedback_state THEN
					pot_to_r04_e_step := 1;
				END_IF;
			1:
				LiquidTransfer_34(sp_time := DINT_TO_TIME(EDTP4S1E_PARA_T2 * 1000),
				sp_accumulation := EDTP4S1E_PARA_AC1,
				done := pot_to_r04_e_step_1_done,
				flowmeter := EDTFQIT1001);
				STFP06.input.auto_run_signal := LiquidTransfer_34.run;
				IF pot_to_r04_e_step_1_done AND (NOT STFP06.input.run_feedback) AND (NOT STFP06.input.auto_run_signal) THEN
					pot_to_r04_e_step_1_done := FALSE;
					pot_to_r04_e_step := 2;
				END_IF;
			2:
				IF EDTFQIT1001.flowrate <= flowrate_threshold THEN
					pot_to_r04_e_step := 3;
				END_IF;
			3:
				EDTFQV1001E.input.auto_open_signal := FALSE;
				EDTLV1003.input.auto_open_signal := FALSE;
				IF EDTFQV1001E.input.close_feedback_state AND EDTLV1003.input.close_feedback_state THEN
					pot_to_r04_e_step := 0;
					pot_to_r04_e := FALSE;
				END_IF;
		END_CASE;
	END_IF;

	//从V52进料
	IF v52_to_r04_e THEN
		CASE v52_to_r04_e_step OF
			0:
				EDTFQV1001E.input.auto_open_signal := TRUE;
				EDTLV1002.input.auto_open_signal := TRUE;
				IF EDTFQV1001E.input.open_feedback_state AND EDTLV1002.input.open_feedback_state THEN
					v52_to_r04_e_step := 1;
				END_IF;
			1:
				LiquidTransfer_35(sp_time := DINT_TO_TIME(EDTP4S1E_PARA_T3 * 1000),
				sp_accumulation := EDTP4S1E_PARA_AC2,
				done := v52_to_r04_e_step_1_done,
				flowmeter := EDTFQIT1001);
				EDTP16.input.auto_run_signal := LiquidTransfer_35.run;
				IF v52_to_r04_e_step_1_done AND (NOT EDTP16.input.run_feedback) AND (NOT EDTP16.input.auto_run_signal) THEN
					v52_to_r04_e_step_1_done := FALSE;
					v52_to_r04_e_step := 2;
				END_IF;
			2:
				IF EDTFQIT1001.flowrate <= flowrate_threshold THEN
					v52_to_r04_e_step := 3;
				END_IF;
			3:
				EDTFQV1001E.input.auto_open_signal := FALSE;
				EDTLV1002.input.auto_open_signal := FALSE;
				IF EDTFQV1001E.input.close_feedback_state AND EDTLV1002.input.close_feedback_state THEN
					v52_to_r04_e_step := 0;
					v52_to_r04_e := FALSE;
				END_IF;
		END_CASE;
	END_IF;

	//=======================================================================================================
	//人工确认步骤可用
	IF (EDTP4S1E.status.run_state) AND (NOT EDTP4S1E_STEP[EDTP4S1E.status.run_step].done AND ((EDTP4S1E.status.run_step = 1) OR (EDTP4S1E.status.run_step = 4) OR (EDTP4S1E.status.run_step = 7))) THEN
		EDTP4S1E.status.confirm_enable := TRUE;
	ELSE
		EDTP4S1E.status.confirm_enable := FALSE;
	END_IF;
END_ACTION

(* ---- EDTP4S1F_ACTION.st ---- *)
ACTION P4S1F_ACT:
	//设定时间
	FOR i := 0 TO EDTP4S1_STEP_NUM DO
		IF EDTP4S1F_ST[i] < T#5s THEN
			EDTP4S1F_ST[i] := T#5s;
		END_IF;
		EDTP4S1F_STEP[i].set_time := EDTP4S1F_ST[i];
	END_FOR;

	//流程步骤
	ProcessHandleFC(EDTP4S1F,EDTP4S1F_STEP[0],EDTP4S1_STEP_NUM);

	//object 手自动切换
	IF (EDTP4S1F.status.mode <> 0) AND (NOT EDTP4S1F.auto_mode_edge) THEN
		EDTP4S1F.auto_mode_edge := TRUE;
		EDTP4S1F.manual_mode_edge := FALSE;

		EDTXV1011.control.auto_operate := TRUE;
		EDTXV1031.control.auto_operate := TRUE;
		EDTP16.control.auto_operate := TRUE;
		EDTLV1002.control.auto_operate := TRUE;
		STFP06.control.auto_operate := TRUE;
		STFLV0602.control.auto_operate := TRUE;
		STFLV0601.control.auto_operate := TRUE;
		EDTLV1003.control.auto_operate := TRUE;
		EDTFQV1001F.control.auto_operate := TRUE;
		EDTTV1012B.control.auto_operate := TRUE;
		EDTXV1033.control.auto_operate := TRUE;
		EDTXV1028.control.auto_operate := TRUE;
		EDTTV1011A.control.auto_operate := TRUE;
		EDTTV1011B.control.auto_operate := TRUE;
		EDTTV1012A.control.auto_operate := TRUE;
		EDTXV1030.control.auto_operate := TRUE;
		EDTR04F.control.auto_operate := TRUE;
		EDTLV1004F.control.auto_operate := TRUE;
	END_IF;

	IF (EDTP4S1F.status.mode = 0) AND (NOT EDTP4S1F.manual_mode_edge) THEN
		EDTP4S1F.manual_mode_edge := TRUE;
		EDTP4S1F.auto_mode_edge := FALSE;

		EDTXV1011.control.manual_operate := TRUE;
		EDTXV1031.control.manual_operate := TRUE;
		EDTP16.control.manual_operate := TRUE;
		EDTLV1002.control.manual_operate := TRUE;
		STFP06.control.manual_operate := TRUE;
		STFLV0602.control.manual_operate := TRUE;
		STFLV0601.control.manual_operate := TRUE;
		EDTLV1003.control.manual_operate := TRUE;
		EDTFQV1001F.control.manual_operate := TRUE;
		EDTTV1012B.control.manual_operate := TRUE;
		EDTXV1033.control.manual_operate := TRUE;
		EDTXV1028.control.manual_operate := TRUE;
		EDTTV1011A.control.manual_operate := TRUE;
		EDTTV1011B.control.manual_operate := TRUE;
		EDTTV1012A.control.manual_operate := TRUE;
		EDTXV1030.control.manual_operate := TRUE;
		EDTR04F.control.manual_operate := TRUE;
		EDTLV1004F.control.manual_operate := TRUE;
	END_IF;

	//错误信号停机
	EDTP4S1F.input.error_signal := (EDTXV1011.status.valve_status >= 2) OR
	(EDTXV1031.status.valve_status >= 2) OR (EDTP16.status.motor_status >= 2) OR
	(EDTLV1002.status.valve_status >= 2) OR (STFP06.status.motor_status >= 2) OR (STFLV0602.status.valve_status >= 2) OR
	(STFLV0601.status.valve_status >= 2) OR (EDTLV1003.status.valve_status >= 2) OR (EDTFQV1001F.status.valve_status >= 2) OR
	(EDTTV1012B.status.valve_status >= 2) OR (EDTXV1033.status.valve_status >= 2) OR
	(EDTXV1028.status.valve_status >= 2) OR (EDTTV1011A.status.valve_status >= 2) OR (EDTTV1011B.status.valve_status >= 2) OR
	(EDTTV1012A.status.valve_status >= 2) OR (EDTR04F.status.motor_status >= 2) OR (EDTXV1030.status.valve_status >= 2);

	//EDTLV1004F自动补水
	//	IF EDTTIT1011.status.value >= EDTP4S1F_PARA_Temp7 THEN
	//		EDTLV1004F.input.auto_open_signal := TRUE;
	//	ELSIF EDTTIT1011.status.value <= (EDTP4S1F_PARA_Temp7 - EDTP4S1F_PARA_Temp8) THEN
	//		EDTLV1004F.input.auto_open_signal := FALSE;
	//	END_IF;
	IF r04f_water THEN
		CASE r04f_water_step OF
			0:
				EDTLV1004F.control.auto_operate := TRUE;
				r04f_water_step := 1;
			1:
				EDTLV1004F.input.auto_open_signal := TRUE;
				r04f_temp := EDTTIT1011.status.value;
				r04f_water_step := 2;
			2:
				IF r04f_temp - EDTTIT1011.status.value >= EDTP4S1F_PARA_Temp8 THEN
					EDTLV1004F.input.auto_open_signal := FALSE;
					r04f_water_step := 0;
					r04f_water := FALSE;
				END_IF;
		END_CASE;
	END_IF;

	IF EDTP4S1F.status.run_state = 1 THEN
		CASE EDTP4S1F.status.run_step OF
			0:
				IF NOT EDTP4S1F_STEP[0].done THEN
					EDTXV1011.control.auto_operate := TRUE;
					EDTXV1031.control.auto_operate := TRUE;
					EDTP16.control.auto_operate := TRUE;
					EDTLV1002.control.auto_operate := TRUE;
					STFP06.control.auto_operate := TRUE;
					STFLV0602.control.auto_operate := TRUE;
					STFLV0601.control.auto_operate := TRUE;
					EDTLV1003.control.auto_operate := TRUE;
					EDTFQV1001F.control.auto_operate := TRUE;
					EDTTV1012B.control.auto_operate := TRUE;
					EDTXV1033.control.auto_operate := TRUE;
					EDTXV1028.control.auto_operate := TRUE;
					EDTTV1011A.control.auto_operate := TRUE;
					EDTTV1011B.control.auto_operate := TRUE;
					EDTTV1012A.control.auto_operate := TRUE;
					EDTXV1030.control.auto_operate := TRUE;
					EDTR04F.control.auto_operate := TRUE;
					EDTLV1004F.control.auto_operate := TRUE;
					EDTP4S1F_STEP[0].done := TRUE;
				END_IF;
			1:
				//手动进DMSO和纯水
			2:
				EDTTV1011A.input.auto_open_signal := TRUE;
				EDTTV1011B.input.auto_open_signal := TRUE;
				EDTXV1033.input.auto_open_signal := TRUE;
				EDTXV1028.input.auto_open_signal := TRUE;
				EDTR04F.input.auto_run_signal := TRUE;
				EDTTV1012B.input.auto_open_signal := TRUE;
				EDTXV1030.input.auto_open_signal := TRUE;
				IF EDTXV1033.input.open_feedback_state AND EDTXV1028.input.open_feedback_state AND EDTR04F.input.run_feedback
					AND EDTTV1012B.input.open_feedback_state AND EDTXV1030.input.open_feedback_state THEN
					EDTP4S1F_STEP[2].done := TRUE;
				END_IF;
			3:
				CASE p4_step1_3f OF
					0:
						IF NOT EDTP4S1F_STEP[3].done THEN
							p4_step1_3f := 1;
						END_IF;
					1:
						R04F_heat := TRUE;
						p4_step1_3f := 2;
					2:
						IF EDTTIT1011.status.value >= EDTP4S1F_PARA_Temp1 THEN
							EDTTV1012B.input.auto_open_signal := FALSE;
							IF EDTTV1012B.input.close_feedback_state THEN
								EDTTV1012A.input.auto_open_signal := TRUE;
								IF EDTTV1012A.input.open_feedback_state THEN
									p4_step1_3f := 3;
								END_IF;
							END_IF;
						END_IF;
					3:
						TON_84.PT := DINT_TO_TIME(EDTP4S1F_PARA_T4 * 3600 * 1000);
						IF EDTTIT1011.status.value >= EDTP4S1F_PARA_Temp2 THEN
							R04F_heat := FALSE;
							R04F_hold := TRUE;
							TON_84.IN := TRUE;
						END_IF;
						IF TON_84.Q THEN
							TON_84.IN := FALSE;
							p4_step1_3f := 4;
						END_IF;
					4:
						p4_step1_3f := 0;
						EDTP4S1F_STEP[3].done := TRUE;
				END_CASE;
				TON_84();
			4:
				//人工取样,确认反应结束
			5:
				R04F_hold := FALSE;
				EDTTV1011A.input.auto_open_signal := FALSE;
				EDTTV1011B.input.auto_open_signal := FALSE;
				IF EDTTV1011A.input.close_feedback_state AND EDTTV1011B.input.close_feedback_state THEN
					EDTP4S1F_STEP[5].done := TRUE;
				END_IF;
			6:
				IF EDTTIT1011.status.value <= EDTP4S1F_PARA_Temp5 THEN
					//					EDTXV1033.input.auto_open_signal := FALSE;
					//					EDTXV1028.input.auto_open_signal := FALSE;
					EDTTV1012A.input.auto_open_signal := FALSE;
				END_IF;
				IF (*EDTXV1033.input.close_feedback_state AND EDTXV1028.input.close_feedback_state AND *)(NOT EDTR04F.input.run_feedback)
					AND EDTTV1012A.input.close_feedback_state THEN
					EDTP4S1F_STEP[6].done := TRUE;
				END_IF;
			7:
				//转移
			8:
				EDTR04F.input.auto_run_signal := FALSE;
				IF NOT EDTR04F.input.run_feedback THEN
					EDTP4S1F_STEP[8].done := TRUE;
				END_IF;
		END_CASE;
	END_IF;

	Slope_5(value := EDTTIT1011.status.value, sample_time := EDTP4S1F_PARA_T5);

	IF R04F_heat THEN
		IF Slope_5.out <= EDTP4S1F_PARA_Slope1 THEN
			EDTTV1011A.input.auto_open_signal := TRUE;
			EDTTV1011B.input.auto_open_signal := TRUE;
		END_IF;
		IF Slope_5.out > EDTP4S1F_PARA_Slope1 AND Slope_5.out <= EDTP4S1F_PARA_Slope2 THEN
			EDTTV1011A.input.auto_open_signal := TRUE;
			EDTTV1011B.input.auto_open_signal := FALSE;
		END_IF;
		IF Slope_5.out > EDTP4S1F_PARA_Slope2 AND Slope_5.out <= EDTP4S1F_PARA_Slope3 THEN
			EDTTV1011A.input.auto_open_signal := FALSE;
			EDTTV1011B.input.auto_open_signal := TRUE;
		END_IF;
		IF Slope_5.out > EDTP4S1F_PARA_Slope3 THEN
			EDTTV1011A.input.auto_open_signal := FALSE;
			EDTTV1011B.input.auto_open_signal := FALSE;
		END_IF;
	END_IF;

	//155-158 大  158-162小阀 162都关
	IF R04F_hold THEN
		IF EDTTIT1011.status.value < EDTP4S1F_PARA_Temp2 THEN
			EDTTV1011A.input.auto_open_signal := TRUE;
			EDTTV1011B.input.auto_open_signal := TRUE;
		END_IF;
		IF EDTTIT1011.status.value < EDTP4S1F_PARA_Temp3 AND EDTTIT1011.status.value >= (EDTP4S1F_PARA_Temp2 + EDTP4S1F_PARA_Temp6) THEN
			EDTTV1011A.input.auto_open_signal := TRUE;
			EDTTV1011B.input.auto_open_signal := FALSE;
		END_IF;
		IF EDTTIT1011.status.value < EDTP4S1F_PARA_Temp4 AND EDTTIT1011.status.value >= (EDTP4S1F_PARA_Temp3 + EDTP4S1F_PARA_Temp6) THEN
			EDTTV1011A.input.auto_open_signal := FALSE;
			EDTTV1011B.input.auto_open_signal := TRUE;
		END_IF;
		IF EDTTIT1011.status.value >= (EDTP4S1F_PARA_Temp4 + EDTP4S1F_PARA_Temp6) THEN
			EDTTV1011A.input.auto_open_signal := FALSE;
			EDTTV1011B.input.auto_open_signal := FALSE;
		END_IF;
	END_IF;

	//======================================================================================================
	//DMSO进料
	//从罐区进料
	IF pot_to_r04_f THEN
		CASE pot_to_r04_f_step OF
			0:
				EDTFQV1001F.input.auto_open_signal := TRUE;
				EDTLV1003.input.auto_open_signal := TRUE;
				STFLV0601.input.auto_open_signal := FALSE;
				STFLV0602.input.auto_open_signal := FALSE;
				IF EDTFQV1001F.input.open_feedback_state AND EDTLV1003.input.open_feedback_state AND
					STFLV0601.input.close_feedback_state AND STFLV0602.input.close_feedback_state THEN
					pot_to_r04_f_step := 1;
				END_IF;
			1:
				LiquidTransfer_36(sp_time := DINT_TO_TIME(EDTP4S1F_PARA_T2 * 1000),
				sp_accumulation := EDTP4S1F_PARA_AC1,
				done := pot_to_r04_f_step_1_done,
				flowmeter := EDTFQIT1001);
				STFP06.input.auto_run_signal := LiquidTransfer_36.run;
				IF pot_to_r04_f_step_1_done AND (NOT STFP06.input.run_feedback) AND (NOT STFP06.input.auto_run_signal) THEN
					pot_to_r04_f_step_1_done := FALSE;
					pot_to_r04_f_step := 2;
				END_IF;
			2:
				IF EDTFQIT1001.flowrate <= flowrate_threshold THEN
					pot_to_r04_f_step := 3;
				END_IF;
			3:
				EDTFQV1001F.input.auto_open_signal := FALSE;
				EDTLV1003.input.auto_open_signal := FALSE;
				IF EDTFQV1001F.input.close_feedback_state AND EDTLV1003.input.close_feedback_state THEN
					pot_to_r04_f_step := 0;
					pot_to_r04_f := FALSE;
				END_IF;
		END_CASE;
	END_IF;

	//从V52进料
	IF v52_to_r04_f THEN
		CASE v52_to_r04_f_step OF
			0:
				EDTFQV1001F.input.auto_open_signal := TRUE;
				EDTLV1002.input.auto_open_signal := TRUE;
				IF EDTFQV1001F.input.open_feedback_state AND EDTLV1002.input.open_feedback_state THEN
					v52_to_r04_f_step := 1;
				END_IF;
			1:
				LiquidTransfer_37(sp_time := DINT_TO_TIME(EDTP4S1F_PARA_T3 * 1000),
				sp_accumulation := EDTP4S1F_PARA_AC2,
				done := v52_to_r04_f_step_1_done,
				flowmeter := EDTFQIT1001);
				EDTP16.input.auto_run_signal := LiquidTransfer_37.run;
				IF v52_to_r04_f_step_1_done AND (NOT EDTP16.input.run_feedback) AND (NOT EDTP16.input.auto_run_signal) THEN
					v52_to_r04_f_step_1_done := FALSE;
					v52_to_r04_f_step := 2;
				END_IF;
			2:
				IF EDTFQIT1001.flowrate <= flowrate_threshold THEN
					v52_to_r04_f_step := 3;
				END_IF;
			3:
				EDTFQV1001F.input.auto_open_signal := FALSE;
				EDTLV1002.input.auto_open_signal := FALSE;
				IF EDTFQV1001F.input.close_feedback_state AND EDTLV1002.input.close_feedback_state THEN
					v52_to_r04_f_step := 0;
					v52_to_r04_f := FALSE;
				END_IF;
		END_CASE;
	END_IF;

	//=======================================================================================================
	//人工确认步骤可用
	IF (EDTP4S1F.status.run_state) AND (NOT EDTP4S1F_STEP[EDTP4S1F.status.run_step].done AND ((EDTP4S1F.status.run_step = 1) OR (EDTP4S1F.status.run_step = 4) OR (EDTP4S1F.status.run_step = 7))) THEN
		EDTP4S1F.status.confirm_enable := TRUE;
	ELSE
		EDTP4S1F.status.confirm_enable := FALSE;
	END_IF;
END_ACTION

(* ---- EDTP4S2A_ACTION.st ---- *)
ACTION P4S2A_ACT:
	//设定时间
	FOR i := 0 TO EDTP4S2_STEP_NUM DO
		IF EDTP4S2A_ST[i] < T#5s THEN
			EDTP4S2A_ST[i] := T#5s;
		END_IF;
		EDTP4S2A_STEP[i].set_time := EDTP4S2A_ST[i];
	END_FOR;

	//流程步骤
	ProcessHandleFC(EDTP4S2A,EDTP4S2A_STEP[0],EDTP4S2_STEP_NUM);

	//object 手自动切换
	IF (EDTP4S2A.status.mode <> 0) AND (NOT EDTP4S2A.auto_mode_edge) THEN
		EDTP4S2A.auto_mode_edge := TRUE;
		EDTP4S2A.manual_mode_edge := FALSE;

		EDTXV1114.control.auto_operate := TRUE;
		EDTR10A.control.auto_operate := TRUE;
		EDTXV1104.control.auto_operate := TRUE;
		EDTXV1109.control.auto_operate := TRUE;
		EDTXV1120.control.auto_operate := TRUE;
		EDTXV1106.control.auto_operate := TRUE;
		EDTFVT1101.control.auto_operate := TRUE;
		EDTTV1101C.control.auto_operate := TRUE;
		EDTTV1101D.control.auto_operate := TRUE;
		EDTTV1101E.control.auto_operate := TRUE;
		EDTTV1101F.control.auto_operate := TRUE;
		EDTXV1107.control.auto_operate := TRUE;
		EDTTV1101A.control.auto_operate := TRUE;
		EDTTV1101B.control.auto_operate := TRUE;
		EDTXV1105.control.auto_operate := TRUE;
		EDTXV1108.control.auto_operate := TRUE;
		EDTTVT1103.control.auto_operate := TRUE;
		EDTFQV1101A.control.auto_operate := TRUE;
		EDTP15.control.auto_operate := TRUE;
	END_IF;

	IF (EDTP4S2A.status.mode = 0) AND (NOT EDTP4S2A.manual_mode_edge) THEN
		EDTP4S2A.manual_mode_edge := TRUE;
		EDTP4S2A.auto_mode_edge := FALSE;

		EDTXV1114.control.manual_operate := TRUE;
		EDTR10A.control.manual_operate := TRUE;
		EDTXV1104.control.manual_operate := TRUE;
		EDTXV1109.control.manual_operate := TRUE;
		EDTXV1120.control.manual_operate := TRUE;
		EDTXV1106.control.manual_operate := TRUE;
		EDTFVT1101.control.manual_operate := TRUE;
		EDTTV1101C.control.manual_operate := TRUE;
		EDTTV1101D.control.manual_operate := TRUE;
		EDTTV1101E.control.manual_operate := TRUE;
		EDTTV1101F.control.manual_operate := TRUE;
		EDTXV1107.control.manual_operate := TRUE;
		EDTTV1101A.control.manual_operate := TRUE;
		EDTTV1101B.control.manual_operate := TRUE;
		EDTXV1105.control.manual_operate := TRUE;
		EDTXV1108.control.manual_operate := TRUE;
		EDTTVT1103.control.manual_operate := TRUE;
		EDTFQV1101A.control.manual_operate := TRUE;
		EDTP15.control.manual_operate := TRUE;
	END_IF;

	//错误信号停机
	EDTP4S2A.input.error_signal :=
	(EDTXV1114.status.valve_status >= 2) OR
	(EDTR10A.status.motor_status >= 2) OR (EDTXV1104.status.valve_status >= 2) OR (EDTXV1109.status.valve_status >= 2) OR
	(EDTXV1120.status.valve_status >= 2) OR (EDTXV1106.status.valve_status >= 2) OR
	(EDTTV1101C.status.valve_status >= 2) OR (EDTTV1101D.status.valve_status >= 2) OR (EDTTV1101E.status.valve_status >= 2) OR
	(EDTTV1101F.status.valve_status >= 2) OR (EDTXV1107.status.valve_status >= 2) OR (EDTTV1101A.status.valve_status >= 2) OR
	(EDTTV1101B.status.valve_status >= 2) OR (EDTXV1105.status.valve_status >= 2) OR (EDTXV1108.status.valve_status >= 2) OR
	(EDTFQV1101A.status.valve_status >= 2) OR (EDTP15.status.motor_status >= 2);

	IF EDTP4S2A.status.run_state = 1 THEN
		CASE EDTP4S2A.status.run_step OF
			0:
				//初始化
				IF NOT EDTP4S2A_STEP[0].done THEN
					EDTXV1114.control.auto_operate := TRUE;
					EDTR10A.control.auto_operate := TRUE;
					EDTXV1104.control.auto_operate := TRUE;
					EDTXV1109.control.auto_operate := TRUE;
					EDTXV1120.control.auto_operate := TRUE;
					EDTXV1106.control.auto_operate := TRUE;
					EDTFVT1101.control.auto_operate := TRUE;
					EDTTV1101C.control.auto_operate := TRUE;
					EDTTV1101D.control.auto_operate := TRUE;
					EDTTV1101E.control.auto_operate := TRUE;
					EDTTV1101F.control.auto_operate := TRUE;
					EDTXV1107.control.auto_operate := TRUE;
					EDTTV1101A.control.auto_operate := TRUE;
					EDTTV1101B.control.auto_operate := TRUE;
					EDTXV1105.control.auto_operate := TRUE;
					EDTXV1108.control.auto_operate := TRUE;
					EDTTVT1103.control.auto_operate := TRUE;
					EDTFQV1101A.control.auto_operate := TRUE;
					EDTP15.control.auto_operate := TRUE;
					EDTP4S2A_STEP[0].done := TRUE;
				END_IF;
			1:
				//准备
				MTBasicsPID_1.Enable := FALSE;
				MTBasicsPID_10.Enable := FALSE;
				EDTXV1114.input.auto_open_signal := FALSE;
				EDTFVT1101.input.auto_degree_set := 100.0;
				EDTTVT1103.input.auto_degree_set := 100.0;
				EDTR10A.input.auto_run_signal := TRUE;
				EDTXV1120.input.auto_open_signal := TRUE;
				IF EDTXV1120.input.open_feedback_state THEN
					EDTXV1104.input.auto_open_signal := TRUE;
				END_IF;
				IF EDTXV1104.input.open_feedback_state THEN
					EDTXV1106.input.auto_open_signal := TRUE;
				END_IF;
				IF EDTXV1106.input.open_feedback_state THEN
					EDTXV1109.input.auto_open_signal := TRUE;
				END_IF;
				IF EDTTIT1101.status.value <= EDTP4S2_PARA_Temp4 THEN
					EDTTV1101A.input.auto_open_signal := FALSE;
					EDTTV1101B.input.auto_open_signal := FALSE;
					IF EDTR10A.input.run_feedback AND EDTXV1104.input.open_feedback_state AND EDTXV1109.input.open_feedback_state AND EDTTV1101A.input.close_feedback_state
						AND EDTTV1101B.input.close_feedback_state AND EDTXV1120.input.open_feedback_state AND EDTXV1106.input.open_feedback_state AND EDTXV1114.input.close_feedback_state
						AND EDTXV1114.input.close_feedback_state THEN
						EDTP4S2A_STEP[1].done := TRUE;
					END_IF;
				ELSIF EDTTIT1101.status.value >= EDTP4S2_PARA_Temp6 THEN
					EDTTV1101A.input.auto_open_signal := TRUE;
					EDTTV1101B.input.auto_open_signal := TRUE;
				END_IF;
			2:
				//启动一级真空泵
			3:
				CASE p4_step2_3a OF
					0:
						IF NOT EDTP4S2A_STEP[3].done THEN
							p4_step2_3a := 1;
						END_IF;
					1:
						HeatPot_3(ST1 := DINT_TO_TIME(EDTP4S2_PARA_T1 * 1000),
						ST2 := DINT_TO_TIME(EDTP4S2_PARA_T2 * 1000),
						V3 := EDTTV1101C,
						V4 := EDTTV1101D,
						V5 := EDTTV1101E,
						V6 := EDTTV1101F,
						done := p4_step2_3a_1_done);
						IF p4_step2_3a_1_done THEN
							p4_step2_3a_1_done := FALSE;
							p4_step2_3a := 2;
						END_IF;
					2:
						IF EDTTIT1101.status.value >= EDTP4S2_PARA_Temp1 THEN
							EDTTV1101C.input.auto_open_signal := FALSE;
						END_IF;
						IF EDTTV1101C.input.close_feedback_state THEN
							p4_step2_3a := 3;
						END_IF;
					3:
						IF EDTTIT1101.status.value >= EDTP4S2_PARA_Temp2 THEN
							p4_step2_3a := 0;
							EDTP4S2A_STEP[3].done := TRUE;
						END_IF;
				END_CASE;
			4:
				//启动二三四级真空泵
			5:
				CASE p4_step2_5a OF
					0:
						IF NOT EDTP4S2A_STEP[5].done THEN
							p4_step2_5a := 1;
						END_IF;
					1:
						IF EDTTIT1102.status.value >= EDTP4S2_PARA_Temp5 THEN
							MTBasicsPID_1.Enable := TRUE;
							MTBasicsPID_10.Enable := FALSE;
							EDTFVT1101.input.auto_degree_set := 0.0;
							p4_step2_5a := 2;
						END_IF;
					2:
						TON_43.PT := DINT_TO_TIME(EDTP4S2_PARA_T3 * 60 * 1000);
						TON_43.IN := TRUE;
						IF TON_43.Q THEN
							TON_43.IN := FALSE;
							p4_step2_5a := 3;
						END_IF;
					3:
						MTBasicsPID_10.Enable := TRUE;
						p4_step2_5a := 4;
					4:
						TON_43.PT := DINT_TO_TIME(EDTP4S2_PARA_T4 * 3600 * 1000);
						TON_43.IN := TRUE;
						IF TON_43.Q THEN
							TON_43.IN := FALSE;
							p4_step2_5a := 5;
							p4_step2_5a_confirm_enable := TRUE;
						END_IF;
					5:
						IF EDTP4S2A_STEP[5].done THEN
							p4_step2_5a := 0;
							p4_step2_5a_confirm_enable := FALSE;
						END_IF;
				END_CASE;
				TON_43();
			6:
				EDTXV1120.input.auto_open_signal := FALSE;
				TON_7.PT := DINT_TO_TIME(EDTP4S2_PARA_T5 * 3600 * 1000);
				IF EDTXV1120.input.close_feedback_state THEN
					EDTXV1107.input.auto_open_signal := TRUE;
					IF EDTXV1107.input.open_feedback_state THEN
						TON_7.IN := TRUE;
					END_IF;
				END_IF;
				IF TON_7.Q THEN
					TON_7.IN := FALSE;
					EDTP4S2A_STEP[6].done := TRUE;
				END_IF;
				TON_7();
			7:
				//观察
			8:
				CASE p4_step2_7a OF
					0:
						IF NOT EDTP4S2A_STEP[8].done THEN
							p4_step2_7a := 1;
						END_IF;
					1:
						CoolPot_4(
							time := cool_pot_time,
							V1 := EDTTV1101A,
							V2 := EDTTV1101B,
							V3 := EDTTV1101F,
							V4 := EDTTV1101D,
							V5 := EDTTV1101E,
							done := p4_step2_7a_1_done);
						IF p4_step2_7a_1_done THEN
							p4_step2_7a_1_done := FALSE;
							p4_step2_7a := 2;
						END_IF;
					2:
						IF EDTTIT1101.status.value <= EDTP4S2_PARA_Temp3 THEN
							p4_step2_7a := 0;
							EDTP4S2A_STEP[8].done := TRUE;
						END_IF;
				END_CASE;
			9:
				//依次关闭四三二级真空泵
			10:
				MTBasicsPID_10.Enable := FALSE;
				EDTFVT1101.input.auto_degree_set := 100.0;
				EDTXV1105.input.auto_open_signal := TRUE;
				EDTXV1108.input.auto_open_signal := TRUE;
				IF EDTPIT1101.status.value >= EDTP4S2_PARA_P1 THEN
					EDTTV1101A.input.auto_open_signal := FALSE;
					EDTTV1101B.input.auto_open_signal := FALSE;
					IF EDTTV1101A.input.close_feedback_state AND EDTTV1101B.input.close_feedback_state THEN
						EDTP4S2A_STEP[10].done := TRUE;
					END_IF;
				END_IF;
			11:
				//关闭一级泵
			12:
				IF EDTPIT1101.status.value >= EDTP4S2_PARA_P2 THEN
					EDTXV1105.input.auto_open_signal := FALSE;
					EDTXV1108.input.auto_open_signal := FALSE;
					EDTP4S2A_STEP[12].done := TRUE;
				END_IF;
			13:
				MTBasicsPID_1.Enable := FALSE;
				EDTTVT1103.input.auto_degree_set := 100.0;
				EDTXV1107.input.auto_open_signal := FALSE;
				EDTXV1114.input.auto_open_signal := TRUE;
				IF EDTXV1107.input.close_feedback_state THEN
					EDTXV1120.input.auto_open_signal := TRUE;
				END_IF;
				IF EDTXV1107.input.close_feedback_state AND EDTXV1114.input.open_feedback_state AND EDTXV1120.input.open_feedback_state THEN
					EDTP4S2A_STEP[13].done := TRUE;
				END_IF;
		END_CASE;
	END_IF;

	//pid调节
	R_TRIG_4(CLK := EDTTVT1103.status.auto_mode);
	IF R_TRIG_4.Q THEN
		MTBasicsPID_1.Enable := TRUE;
	END_IF;
	F_TRIG_4(CLK := EDTTVT1103.status.auto_mode);
	IF F_TRIG_4.Q THEN
		MTBasicsPID_1.Enable := FALSE;
	END_IF;

	//	MTBasicsPID_1.Enable := TRUE;
	MTBasicsPID_1.Invert := TRUE;
	MTBasicsPID_1.PIDParameters.Gain := EDTPid1103Para.gain;
	MTBasicsPID_1.PIDParameters.IntegrationTime := EDTPid1103Para.integration_time;
	MTBasicsPID_1.PIDParameters.DerivativeTime := EDTPid1103Para.derivative_time;
	MTBasicsPID_1.MinOut := 0.0;
	MTBasicsPID_1.MaxOut := 100.0;
	MTBasicsPID_1.ActValue := EDTTIT1103.status.value;
	MTBasicsPID_1.SetValue := EDTPid1103Para.set_value;
	MTBasicsPID_1.Update := EDTPid1103.update;
	MTBasicsPID_1();
	EDTPid1103.out := MTBasicsPID_1.Out;
	IF MTBasicsPID_1.Active THEN
		EDTTVT1103.input.auto_degree_set := MTBasicsPID_1.Out;
		//	ELSE
		//		EDTTVT1103.input.auto_degree_set := 0.0;
	END_IF;
	IF MTBasicsPID_1.UpdateDone THEN
		EDTPid1103.update := FALSE;
	END_IF;

	//FVT1101 pid调节
	R_TRIG_5(CLK := EDTFVT1101.status.auto_mode);
	IF R_TRIG_5.Q THEN
		MTBasicsPID_10.Enable := TRUE;
	END_IF;
	F_TRIG_5(CLK := EDTFVT1101.status.auto_mode);
	IF F_TRIG_5.Q THEN
		MTBasicsPID_10.Enable := FALSE;
	END_IF;

	//	MTBasicsPID_10.Enable := TRUE;
	MTBasicsPID_10.PIDParameters.Gain := EDTPidFVT1101Para.gain;
	MTBasicsPID_10.PIDParameters.IntegrationTime := EDTPidFVT1101Para.integration_time;
	MTBasicsPID_10.PIDParameters.DerivativeTime := EDTPidFVT1101Para.derivative_time;
	MTBasicsPID_10.MinOut := 0.0;
	MTBasicsPID_10.MaxOut := 100.0;
	MTBasicsPID_10.SetValue := EDTPidFVT1101Para.set_value;
	MTBasicsPID_10.ActValue := EDTFIT1101.flowrate;
	MTBasicsPID_10.Update := EDTPidFVT1101.update;
	MTBasicsPID_10();
	EDTPidFVT1101.out := MTBasicsPID_10.Out;
	IF MTBasicsPID_10.Active THEN
		EDTFVT1101.input.auto_degree_set := MTBasicsPID_10.Out + EDTPidFVT1101Para.min_out;
		//	ELSE
		//		EDTFVT1101.input.auto_degree_set := 0.0;
	END_IF;
	IF MTBasicsPID_10.UpdateDone THEN
		EDTPidFVT1101.update := FALSE;
	END_IF;

	//人工确认步骤可用
	IF (EDTP4S2A.status.run_state) AND (NOT EDTP4S2A_STEP[EDTP4S2A.status.run_step].done AND ((EDTP4S2A.status.run_step = 2) OR (EDTP4S2A.status.run_step = 4) OR (EDTP4S2A.status.run_step = 7)
		OR (EDTP4S2A.status.run_step = 9) OR (EDTP4S2A.status.run_step = 11) OR (p4_step2_5a_confirm_enable))) THEN
		EDTP4S2A.status.confirm_enable := TRUE;
	ELSE
		EDTP4S2A.status.confirm_enable := FALSE;
	END_IF;
END_ACTION

(* ---- EDTP4S2B_ACTION.st ---- *)
ACTION P4S2B_ACT:
		//设定时间
	FOR i := 0 TO EDTP4S2_STEP_NUM DO
		IF EDTP4S2B_ST[i] < T#5s THEN
			EDTP4S2B_ST[i] := T#5s;
		END_IF;
		EDTP4S2B_STEP[i].set_time := EDTP4S2B_ST[i];
	END_FOR;

	//流程步骤
	ProcessHandleFC(EDTP4S2B,EDTP4S2B_STEP[0],EDTP4S2_STEP_NUM);

	//object 手自动切换
	IF (EDTP4S2B.status.mode <> 0) AND (NOT EDTP4S2B.auto_mode_edge) THEN
		EDTP4S2B.auto_mode_edge := TRUE;
		EDTP4S2B.manual_mode_edge := FALSE;

		EDTXV1132.control.auto_operate := TRUE;
		EDTR10B.control.auto_operate := TRUE;
		EDTXV1124.control.auto_operate := TRUE;
		EDTXV1129.control.auto_operate := TRUE;
		EDTXV1136.control.auto_operate := TRUE;
		EDTXV1126.control.auto_operate := TRUE;
		EDTFVT1103.control.auto_operate := TRUE;
		EDTTV1104C.control.auto_operate := TRUE;
		EDTTV1104D.control.auto_operate := TRUE;
		EDTTV1104E.control.auto_operate := TRUE;
		EDTTV1104F.control.auto_operate := TRUE;
		EDTXV1127.control.auto_operate := TRUE;
		EDTTV1104A.control.auto_operate := TRUE;
		EDTTV1104B.control.auto_operate := TRUE;
		EDTXV1125.control.auto_operate := TRUE;
		EDTXV1128.control.auto_operate := TRUE;
		EDTTVT1106.control.auto_operate := TRUE;
		EDTFQV1101B.control.auto_operate := TRUE;
		EDTP15.control.auto_operate := TRUE;
	END_IF;

	IF (EDTP4S2B.status.mode = 0) AND (NOT EDTP4S2B.manual_mode_edge) THEN
		EDTP4S2B.manual_mode_edge := TRUE;
		EDTP4S2B.auto_mode_edge := FALSE;

		EDTXV1132.control.manual_operate := TRUE;
		EDTR10B.control.manual_operate := TRUE;
		EDTXV1124.control.manual_operate := TRUE;
		EDTXV1129.control.manual_operate := TRUE;
		EDTXV1136.control.manual_operate := TRUE;
		EDTXV1126.control.manual_operate := TRUE;
		EDTFVT1103.control.manual_operate := TRUE;
		EDTTV1104C.control.manual_operate := TRUE;
		EDTTV1104D.control.manual_operate := TRUE;
		EDTTV1104E.control.manual_operate := TRUE;
		EDTTV1104F.control.manual_operate := TRUE;
		EDTXV1127.control.manual_operate := TRUE;
		EDTTV1104A.control.manual_operate := TRUE;
		EDTTV1104B.control.manual_operate := TRUE;
		EDTXV1125.control.manual_operate := TRUE;
		EDTXV1128.control.manual_operate := TRUE;
		EDTTVT1106.control.manual_operate := TRUE;
		EDTFQV1101B.control.manual_operate := TRUE;
		EDTP15.control.manual_operate := TRUE;
	END_IF;

	//错误信号停机
	EDTP4S2B.input.error_signal :=
	(EDTXV1132.status.valve_status >= 2) OR
	(EDTR10B.status.motor_status >= 2) OR (EDTXV1124.status.valve_status >= 2) OR (EDTXV1129.status.valve_status >= 2) OR
	(EDTXV1136.status.valve_status >= 2) OR (EDTXV1126.status.valve_status >= 2) OR
	(EDTTV1104C.status.valve_status >= 2) OR (EDTTV1104D.status.valve_status >= 2) OR (EDTTV1104E.status.valve_status >= 2) OR
	(EDTTV1104F.status.valve_status >= 2) OR (EDTXV1127.status.valve_status >= 2) OR (EDTTV1104A.status.valve_status >= 2) OR
	(EDTTV1104B.status.valve_status >= 2) OR (EDTXV1125.status.valve_status >= 2) OR (EDTXV1128.status.valve_status >= 2) OR
	(EDTFQV1101B.status.valve_status >= 2) OR (EDTP15.status.motor_status >= 2);

	IF EDTP4S2B.status.run_state = 1 THEN
		CASE EDTP4S2B.status.run_step OF
			0:
				//初始化
				IF NOT EDTP4S2B_STEP[0].done THEN
					EDTXV1132.control.auto_operate := TRUE;
					EDTR10B.control.auto_operate := TRUE;
					EDTXV1124.control.auto_operate := TRUE;
					EDTXV1129.control.auto_operate := TRUE;
					EDTXV1136.control.auto_operate := TRUE;
					EDTXV1126.control.auto_operate := TRUE;
					EDTFVT1103.control.auto_operate := TRUE;
					EDTTV1104C.control.auto_operate := TRUE;
					EDTTV1104D.control.auto_operate := TRUE;
					EDTTV1104E.control.auto_operate := TRUE;
					EDTTV1104F.control.auto_operate := TRUE;
					EDTXV1127.control.auto_operate := TRUE;
					EDTTV1104A.control.auto_operate := TRUE;
					EDTTV1104B.control.auto_operate := TRUE;
					EDTXV1125.control.auto_operate := TRUE;
					EDTXV1128.control.auto_operate := TRUE;
					EDTTVT1106.control.auto_operate := TRUE;
					EDTFQV1101B.control.auto_operate := TRUE;
					EDTP15.control.auto_operate := TRUE;
					EDTP4S2B_STEP[0].done := TRUE;
				END_IF;
			1:
				//准备
				MTBasicsPID_5.Enable := FALSE;
				MTBasicsPID_11.Enable := FALSE;
				EDTXV1132.input.auto_open_signal := FALSE;
				EDTFVT1103.input.auto_degree_set := 100.0;
				EDTTVT1106.input.auto_degree_set := 100.0;
				EDTR10B.input.auto_run_signal := TRUE;
				EDTXV1136.input.auto_open_signal := TRUE;
				IF EDTXV1136.input.open_feedback_state THEN
					EDTXV1124.input.auto_open_signal := TRUE;
				END_IF;
				IF EDTXV1124.input.open_feedback_state THEN
					EDTXV1126.input.auto_open_signal := TRUE;
				END_IF;
				IF EDTXV1126.input.open_feedback_state THEN
					EDTXV1129.input.auto_open_signal := TRUE;
				END_IF;
				IF EDTTIT1104.status.value <= EDTP4S2_PARA_Temp4 THEN
					EDTTV1104A.input.auto_open_signal := FALSE;
					EDTTV1104B.input.auto_open_signal := FALSE;
					IF EDTR10B.input.run_feedback AND EDTXV1124.input.open_feedback_state AND EDTXV1129.input.open_feedback_state AND EDTTV1104A.input.close_feedback_state
						AND EDTTV1104B.input.close_feedback_state AND EDTXV1136.input.open_feedback_state AND EDTXV1126.input.open_feedback_state AND EDTXV1132.input.close_feedback_state
						AND EDTXV1132.input.close_feedback_state THEN
						EDTP4S2B_STEP[1].done := TRUE;
					END_IF;
				ELSIF EDTTIT1104.status.value >=  (EDTP4S2_PARA_Temp4 + 1) THEN
					EDTTV1104A.input.auto_open_signal := TRUE;
					EDTTV1104B.input.auto_open_signal := TRUE;
				END_IF;
			2:
				//启动一级真空泵
			3:
				CASE p4_step2_3b OF
					0:
						IF NOT EDTP4S2B_STEP[3].done THEN
							p4_step2_3b := 1;
						END_IF;
					1:
						HeatPot_12(ST1 := DINT_TO_TIME(EDTP4S2_PARA_T1 * 1000),
						ST2 := DINT_TO_TIME(EDTP4S2_PARA_T2 * 1000),
						V3 := EDTTV1104C,
						V4 := EDTTV1104D,
						V5 := EDTTV1104E,
						V6 := EDTTV1104F,
						done := p4_step2_3b_1_done);
						IF p4_step2_3b_1_done THEN
							p4_step2_3b_1_done := FALSE;
							p4_step2_3b := 2;
						END_IF;
					2:
						IF EDTTIT1104.status.value >= EDTP4S2_PARA_Temp1 THEN
							EDTTV1104C.input.auto_open_signal := FALSE;
						END_IF;
						IF EDTTV1104C.input.close_feedback_state THEN
							p4_step2_3b := 3;
						END_IF;
					3:
						IF EDTTIT1104.status.value >= EDTP4S2_PARA_Temp2 THEN
							p4_step2_3b := 0;
							EDTP4S2B_STEP[3].done := TRUE;
						END_IF;
				END_CASE;
			4:
				//启动二三四级真空泵
			5:
				CASE p4_step2_5b OF
					0:
						IF NOT EDTP4S2B_STEP[5].done THEN
							p4_step2_5b := 1;
						END_IF;
					1:
						IF EDTTIT1105.status.value >= EDTP4S2_PARA_Temp5 THEN
							MTBasicsPID_5.Enable := TRUE;
							MTBasicsPID_11.Enable := FALSE;
							EDTFVT1103.input.auto_degree_set := 0.0;
							p4_step2_5b := 2;
						END_IF;
					2:
						TON_64.PT := DINT_TO_TIME(EDTP4S2_PARA_T3 * 60 * 1000);
						TON_64.IN := TRUE;
						IF TON_64.Q THEN
							TON_64.IN := FALSE;
							p4_step2_5b := 3;
						END_IF;
					3:
						MTBasicsPID_11.Enable := TRUE;
						p4_step2_5b := 4;
					4:
						TON_64.PT := DINT_TO_TIME(EDTP4S2_PARA_T4 * 3600 * 1000);
						TON_64.IN := TRUE;
						IF TON_64.Q THEN
							TON_64.IN := FALSE;
							p4_step2_5b_confirm_enable := TRUE;
							p4_step2_5b := 5;
						END_IF;
					5:
						IF EDTP4S2B_STEP[5].done THEN
							p4_step2_5b := 0;
							p4_step2_5b_confirm_enable := FALSE;
						END_IF;
				END_CASE;
				TON_64();
			6:
				EDTXV1136.input.auto_open_signal := FALSE;
				TON_13.PT := DINT_TO_TIME(EDTP4S2_PARA_T5 * 3600 * 1000);
				IF EDTXV1136.input.close_feedback_state THEN
					EDTXV1127.input.auto_open_signal := TRUE;
					IF EDTXV1127.input.open_feedback_state THEN
						TON_13.IN := TRUE;
					END_IF;
				END_IF;
				IF TON_13.Q THEN
					TON_13.IN := FALSE;
					EDTP4S2B_STEP[6].done := TRUE;
				END_IF;
				TON_13();
			7:
				//观察
			8:
				CASE p4_step2_7b OF
					0:
						IF NOT EDTP4S2B_STEP[8].done THEN
							p4_step2_7b := 1;
						END_IF;
					1:
						CoolPot_1(
							time := cool_pot_time,
							V1 := EDTTV1104A,
							V2 := EDTTV1104B,
							V3 := EDTTV1104F,
							V4 := EDTTV1104D,
							V5 := EDTTV1104E,
							done := p4_step2_7b_1_done);
						IF p4_step2_7b_1_done THEN
							p4_step2_7b_1_done := FALSE;
							p4_step2_7b := 2;
						END_IF;
					2:
						IF EDTTIT1104.status.value <= EDTP4S2_PARA_Temp3 THEN
							p4_step2_7b := 0;
							EDTP4S2B_STEP[8].done := TRUE;
						END_IF;
				END_CASE;
			9:
				//依次关闭四三二级真空泵
			10:
				MTBasicsPID_11.Enable := FALSE;
				EDTFVT1103.input.auto_degree_set := 100.0;
				EDTXV1125.input.auto_open_signal := TRUE;
				EDTXV1128.input.auto_open_signal := TRUE;
				IF EDTPIT1102.status.value >= EDTP4S2_PARA_P1 THEN
					EDTTV1104A.input.auto_open_signal := FALSE;
					EDTTV1104B.input.auto_open_signal := FALSE;
					IF EDTTV1104A.input.close_feedback_state AND EDTTV1104B.input.close_feedback_state THEN
						EDTP4S2B_STEP[10].done := TRUE;
					END_IF;
				END_IF;
			11:
				//关闭一级泵
			12:
				IF EDTPIT1102.status.value >= EDTP4S2_PARA_P2 THEN
					EDTXV1125.input.auto_open_signal := FALSE;
					EDTXV1128.input.auto_open_signal := FALSE;
					EDTP4S2B_STEP[12].done := TRUE;
				END_IF;
			13:
				MTBasicsPID_5.Enable := FALSE;
				EDTTVT1106.input.auto_degree_set := 100.0;
				EDTXV1127.input.auto_open_signal := FALSE;
				EDTXV1132.input.auto_open_signal := TRUE;
				IF EDTXV1127.input.close_feedback_state THEN
					EDTXV1136.input.auto_open_signal := TRUE;
				END_IF;
				IF EDTXV1127.input.close_feedback_state AND EDTXV1132.input.open_feedback_state AND EDTXV1136.input.open_feedback_state THEN
					EDTP4S2B_STEP[13].done := TRUE;
				END_IF;
		END_CASE;
	END_IF;

	//pid调节
	R_TRIG_6(CLK := EDTTVT1106.status.auto_mode);
	IF R_TRIG_6.Q THEN
		MTBasicsPID_5.Enable := TRUE;
	END_IF;
	F_TRIG_6(CLK := EDTTVT1106.status.auto_mode);
	IF F_TRIG_6.Q THEN
		MTBasicsPID_5.Enable := FALSE;
	END_IF;
	//	MTBasicsPID_5.Enable := TRUE;
	MTBasicsPID_5.Invert := TRUE;
	MTBasicsPID_5.PIDParameters.Gain := EDTPid1106Para.gain;
	MTBasicsPID_5.PIDParameters.IntegrationTime := EDTPid1106Para.integration_time;
	MTBasicsPID_5.PIDParameters.DerivativeTime := EDTPid1106Para.derivative_time;
	MTBasicsPID_5.MinOut := 0.0;
	MTBasicsPID_5.MaxOut := 100.0;
	MTBasicsPID_5.ActValue := EDTTIT1106.status.value;
	MTBasicsPID_5.SetValue := EDTPid1106Para.set_value;
	MTBasicsPID_5.Update := EDTPid1106.update;
	MTBasicsPID_5();
	EDTPid1106.out := MTBasicsPID_5.Out;
	IF MTBasicsPID_5.Active THEN
		EDTTVT1106.input.auto_degree_set := MTBasicsPID_5.Out;
		//	ELSE
		//		EDTTVT1106.input.auto_degree_set := 0.0;
	END_IF;
	IF MTBasicsPID_5.UpdateDone THEN
		EDTPid1106.update := FALSE;
	END_IF;

	//FVT1103 pid调节
	R_TRIG_7(CLK := EDTFVT1103.status.auto_mode);
	IF R_TRIG_7.Q THEN
		MTBasicsPID_11.Enable := TRUE;
	END_IF;
	F_TRIG_7(CLK := EDTFVT1103.status.auto_mode);
	IF F_TRIG_7.Q THEN
		MTBasicsPID_11.Enable := FALSE;
	END_IF;
	//	MTBasicsPID_11.Enable := TRUE;
	MTBasicsPID_11.PIDParameters.Gain := EDTPidFVT1103Para.gain;
	MTBasicsPID_11.PIDParameters.IntegrationTime := EDTPidFVT1103Para.integration_time;
	MTBasicsPID_11.PIDParameters.DerivativeTime := EDTPidFVT1103Para.derivative_time;
	MTBasicsPID_11.MinOut := 0.0;
	MTBasicsPID_11.MaxOut := 100.0;
	MTBasicsPID_11.SetValue := EDTPidFVT1103Para.set_value;
	MTBasicsPID_11.ActValue := EDTFIT1103.flowrate;
	MTBasicsPID_11.Update := EDTPidFVT1103.update;
	MTBasicsPID_11();
	EDTPidFVT1103.out := MTBasicsPID_11.Out;
	IF MTBasicsPID_11.Active THEN
		EDTFVT1103.input.auto_degree_set := MTBasicsPID_11.Out + EDTPidFVT1103Para.min_out;
		//	ELSE
		//		EDTFVT1103.input.auto_degree_set := 0.0;
	END_IF;
	IF MTBasicsPID_11.UpdateDone THEN
		EDTPidFVT1103.update := FALSE;
	END_IF;

	//人工确认步骤可用
	IF (EDTP4S2B.status.run_state) AND (NOT EDTP4S2B_STEP[EDTP4S2B.status.run_step].done AND ((EDTP4S2B.status.run_step = 2) OR (EDTP4S2B.status.run_step = 4) OR (EDTP4S2B.status.run_step = 7)
		OR (EDTP4S2B.status.run_step = 9) OR (EDTP4S2B.status.run_step = 11) OR (p4_step2_5b_confirm_enable))) THEN
		EDTP4S2B.status.confirm_enable := TRUE;
	ELSE
		EDTP4S2B.status.confirm_enable := FALSE;
	END_IF;
END_ACTION

(* ---- EDTP4S2C_ACTION.st ---- *)
ACTION P4S2C_ACT:
		//设定时间
	FOR i := 0 TO EDTP4S2_STEP_NUM DO
		IF EDTP4S2C_ST[i] < T#5s THEN
			EDTP4S2C_ST[i] := T#5s;
		END_IF;
		EDTP4S2C_STEP[i].set_time := EDTP4S2C_ST[i];
	END_FOR;

	//流程步骤
	ProcessHandleFC(EDTP4S2C,EDTP4S2C_STEP[0],EDTP4S2_STEP_NUM);

	//object 手自动切换
	IF (EDTP4S2C.status.mode <> 0) AND (NOT EDTP4S2C.auto_mode_edge) THEN
		EDTP4S2C.auto_mode_edge := TRUE;
		EDTP4S2C.manual_mode_edge := FALSE;

		EDTXV1148.control.auto_operate := TRUE;
		EDTR10C.control.auto_operate := TRUE;
		EDTXV1140.control.auto_operate := TRUE;
		EDTXV1145.control.auto_operate := TRUE;
		EDTXV1152.control.auto_operate := TRUE;
		EDTXV1142.control.auto_operate := TRUE;
		EDTFVT1105.control.auto_operate := TRUE;
		EDTTV1107C.control.auto_operate := TRUE;
		EDTTV1107D.control.auto_operate := TRUE;
		EDTTV1107E.control.auto_operate := TRUE;
		EDTTV1107F.control.auto_operate := TRUE;
		EDTXV1143.control.auto_operate := TRUE;
		EDTTV1107A.control.auto_operate := TRUE;
		EDTTV1107B.control.auto_operate := TRUE;
		EDTXV1141.control.auto_operate := TRUE;
		EDTXV1144.control.auto_operate := TRUE;
		EDTTVT1109.control.auto_operate := TRUE;
		EDTFQV1101C.control.auto_operate := TRUE;
		EDTP15.control.auto_operate := TRUE;
	END_IF;

	IF (EDTP4S2C.status.mode = 0) AND (NOT EDTP4S2C.manual_mode_edge) THEN
		EDTP4S2C.manual_mode_edge := TRUE;
		EDTP4S2C.auto_mode_edge := FALSE;

		EDTXV1148.control.manual_operate := TRUE;
		EDTR10C.control.manual_operate := TRUE;
		EDTXV1140.control.manual_operate := TRUE;
		EDTXV1145.control.manual_operate := TRUE;
		EDTXV1152.control.manual_operate := TRUE;
		EDTXV1142.control.manual_operate := TRUE;
		EDTFVT1105.control.manual_operate := TRUE;
		EDTTV1107C.control.manual_operate := TRUE;
		EDTTV1107D.control.manual_operate := TRUE;
		EDTTV1107E.control.manual_operate := TRUE;
		EDTTV1107F.control.manual_operate := TRUE;
		EDTXV1143.control.manual_operate := TRUE;
		EDTTV1107A.control.manual_operate := TRUE;
		EDTTV1107B.control.manual_operate := TRUE;
		EDTXV1141.control.manual_operate := TRUE;
		EDTXV1144.control.manual_operate := TRUE;
		EDTTVT1109.control.manual_operate := TRUE;
		EDTFQV1101C.control.manual_operate := TRUE;
		EDTP15.control.manual_operate := TRUE;
	END_IF;

	//错误信号停机
	EDTP4S2C.input.error_signal :=
	(EDTXV1148.status.valve_status >= 2) OR
	(EDTR10C.status.motor_status >= 2) OR (EDTXV1140.status.valve_status >= 2) OR (EDTXV1145.status.valve_status >= 2) OR
	(EDTXV1152.status.valve_status >= 2) OR (EDTXV1142.status.valve_status >= 2) OR
	(EDTTV1107C.status.valve_status >= 2) OR (EDTTV1107D.status.valve_status >= 2) OR (EDTTV1107E.status.valve_status >= 2) OR
	(EDTTV1107F.status.valve_status >= 2) OR (EDTXV1143.status.valve_status >= 2) OR (EDTTV1107A.status.valve_status >= 2) OR
	(EDTTV1107B.status.valve_status >= 2) OR (EDTXV1141.status.valve_status >= 2) OR (EDTXV1144.status.valve_status >= 2) OR
	(EDTFQV1101C.status.valve_status >= 2) OR (EDTP15.status.motor_status >= 2);

	IF EDTP4S2C.status.run_state = 1 THEN
		CASE EDTP4S2C.status.run_step OF
			0:
				//初始化
				IF NOT EDTP4S2C_STEP[0].done THEN
					EDTXV1148.control.auto_operate := TRUE;
					EDTR10C.control.auto_operate := TRUE;
					EDTXV1140.control.auto_operate := TRUE;
					EDTXV1145.control.auto_operate := TRUE;
					EDTXV1152.control.auto_operate := TRUE;
					EDTXV1142.control.auto_operate := TRUE;
					EDTFVT1105.control.auto_operate := TRUE;
					EDTTV1107C.control.auto_operate := TRUE;
					EDTTV1107D.control.auto_operate := TRUE;
					EDTTV1107E.control.auto_operate := TRUE;
					EDTTV1107F.control.auto_operate := TRUE;
					EDTXV1143.control.auto_operate := TRUE;
					EDTTV1107A.control.auto_operate := TRUE;
					EDTTV1107B.control.auto_operate := TRUE;
					EDTXV1141.control.auto_operate := TRUE;
					EDTXV1144.control.auto_operate := TRUE;
					EDTTVT1109.control.auto_operate := TRUE;
					EDTFQV1101C.control.auto_operate := TRUE;
					EDTP15.control.auto_operate := TRUE;
					EDTP4S2C_STEP[0].done := TRUE;
				END_IF;
			1:
				//准备
				MTBasicsPID_6.Enable := FALSE;
				MTBasicsPID_12.Enable := FALSE;
				EDTXV1148.input.auto_open_signal := FALSE;
				EDTFVT1105.input.auto_degree_set := 100.0;
				EDTTVT1109.input.auto_degree_set := 100.0;
				EDTR10C.input.auto_run_signal := TRUE;
				EDTXV1152.input.auto_open_signal := TRUE;
				IF EDTXV1152.input.open_feedback_state THEN
					EDTXV1140.input.auto_open_signal := TRUE;
				END_IF;
				IF EDTXV1140.input.open_feedback_state THEN
					EDTXV1142.input.auto_open_signal := TRUE;
				END_IF;
				IF EDTXV1142.input.open_feedback_state THEN
					EDTXV1145.input.auto_open_signal := TRUE;
				END_IF;
				IF EDTTIT1107.status.value <= EDTP4S2_PARA_Temp4 THEN
					EDTTV1107A.input.auto_open_signal := FALSE;
					EDTTV1107B.input.auto_open_signal := FALSE;
					IF EDTR10C.input.run_feedback AND EDTXV1140.input.open_feedback_state AND EDTXV1145.input.open_feedback_state AND EDTTV1107A.input.close_feedback_state
						AND EDTTV1107B.input.close_feedback_state AND EDTXV1152.input.open_feedback_state AND EDTXV1142.input.open_feedback_state AND EDTXV1148.input.close_feedback_state
						AND EDTXV1148.input.close_feedback_state THEN
						EDTP4S2C_STEP[1].done := TRUE;
					END_IF;
				ELSIF EDTTIT1107.status.value >=  (EDTP4S2_PARA_Temp4 + 1) THEN
					EDTTV1107A.input.auto_open_signal := TRUE;
					EDTTV1107B.input.auto_open_signal := TRUE;
				END_IF;
			2:
				//启动一级真空泵
			3:
				CASE p4_step2_3c OF
					0:
						IF NOT EDTP4S2C_STEP[3].done THEN
							p4_step2_3c := 1;
						END_IF;
					1:
						HeatPot_14(ST1 := DINT_TO_TIME(EDTP4S2_PARA_T1 * 1000),
						ST2 := DINT_TO_TIME(EDTP4S2_PARA_T2 * 1000),
						V3 := EDTTV1107C,
						V4 := EDTTV1107D,
						V5 := EDTTV1107E,
						V6 := EDTTV1107F,
						done := p4_step2_3c_1_done);
						IF p4_step2_3c_1_done THEN
							p4_step2_3c_1_done := FALSE;
							p4_step2_3c := 2;
						END_IF;
					2:
						IF EDTTIT1107.status.value >= EDTP4S2_PARA_Temp1 THEN
							EDTTV1107C.input.auto_open_signal := FALSE;
						END_IF;
						IF EDTTV1107C.input.close_feedback_state THEN
							p4_step2_3c := 3;
						END_IF;
					3:
						IF EDTTIT1107.status.value >= EDTP4S2_PARA_Temp2 THEN
							p4_step2_3c := 0;
							EDTP4S2C_STEP[3].done := TRUE;
						END_IF;
				END_CASE;
			4:
				//启动二三四级真空泵
			5:
				CASE p4_step2_5c OF
					0:
						IF NOT EDTP4S2C_STEP[5].done THEN
							p4_step2_5c := 1;
						END_IF;
					1:
						IF EDTTIT1108.status.value >= EDTP4S2_PARA_Temp5 THEN
							MTBasicsPID_6.Enable := TRUE;
							MTBasicsPID_12.Enable := FALSE;
							EDTFVT1105.input.auto_degree_set := 0.0;
							p4_step2_5c := 2;
						END_IF;
					2:
						TON_68.PT := DINT_TO_TIME(EDTP4S2_PARA_T3 * 60 * 1000);
						TON_68.IN := TRUE;
						IF TON_68.Q THEN
							TON_68.IN := FALSE;
							p4_step2_5c := 3;
						END_IF;
					3:
						MTBasicsPID_12.Enable := TRUE;
						p4_step2_5c := 4;
					4:
						TON_68.PT := DINT_TO_TIME(EDTP4S2_PARA_T4 * 3600 * 1000);
						TON_68.IN := TRUE;
						IF TON_68.Q THEN
							TON_68.IN := FALSE;
							p4_step2_5c_confirm_enable := TRUE;
							p4_step2_5c := 5;
						END_IF;
					5:
						IF EDTP4S2C_STEP[5].done THEN
							p4_step2_5c_confirm_enable := FALSE;
							p4_step2_5c := 0;
						END_IF;
				END_CASE;
				TON_68();
			6:
				EDTXV1152.input.auto_open_signal := FALSE;
				TON_16.PT := DINT_TO_TIME(EDTP4S2_PARA_T5 * 3600 * 1000);
				IF EDTXV1152.input.close_feedback_state THEN
					EDTXV1143.input.auto_open_signal := TRUE;
					IF EDTXV1143.input.open_feedback_state THEN
						TON_16.IN := TRUE;
					END_IF;
				END_IF;
				IF TON_16.Q THEN
					TON_16.IN := FALSE;
					EDTP4S2C_STEP[6].done := TRUE;
				END_IF;
				TON_16();
			7:
				//观察
			8:
				CASE p4_step2_7c OF
					0:
						IF NOT EDTP4S2C_STEP[8].done THEN
							p4_step2_7c := 1;
						END_IF;
					1:
						CoolPot_2(
							time := cool_pot_time,
							V1 := EDTTV1107A,
							V2 := EDTTV1107B,
							V3 := EDTTV1107F,
							V4 := EDTTV1107D,
							V5 := EDTTV1107E,
							done := p4_step2_7c_1_done);
						IF p4_step2_7c_1_done THEN
							p4_step2_7c_1_done := FALSE;
							p4_step2_7c := 2;
						END_IF;
					2:
						IF EDTTIT1107.status.value <= EDTP4S2_PARA_Temp3 THEN
							p4_step2_7c := 0;
							EDTP4S2C_STEP[8].done := TRUE;
						END_IF;
				END_CASE;
			9:
				//依次关闭四三二级真空泵
			10:
				MTBasicsPID_12.Enable := FALSE;
				EDTFVT1105.input.auto_degree_set := 100.0;
				EDTXV1141.input.auto_open_signal := TRUE;
				EDTXV1144.input.auto_open_signal := TRUE;
				IF EDTPIT1103.status.value >= EDTP4S2_PARA_P1 THEN
					EDTTV1107A.input.auto_open_signal := FALSE;
					EDTTV1107B.input.auto_open_signal := FALSE;
					IF EDTTV1107A.input.close_feedback_state AND EDTTV1107B.input.close_feedback_state THEN
						EDTP4S2C_STEP[10].done := TRUE;
					END_IF;
				END_IF;
			11:
				//关闭一级泵
			12:
				IF EDTPIT1103.status.value >= EDTP4S2_PARA_P2 THEN
					EDTXV1141.input.auto_open_signal := FALSE;
					EDTXV1144.input.auto_open_signal := FALSE;
					EDTP4S2C_STEP[12].done := TRUE;
				END_IF;
			13:
				MTBasicsPID_6.Enable := FALSE;
				EDTTVT1109.input.auto_degree_set := 100.0;
				EDTXV1143.input.auto_open_signal := FALSE;
				EDTXV1148.input.auto_open_signal := TRUE;
				IF EDTXV1143.input.close_feedback_state THEN
					EDTXV1152.input.auto_open_signal := TRUE;
				END_IF;
				IF EDTXV1143.input.close_feedback_state AND EDTXV1148.input.open_feedback_state AND EDTXV1152.input.open_feedback_state THEN
					EDTP4S2C_STEP[13].done := TRUE;
				END_IF;
		END_CASE;
	END_IF;

	//pid调节
	R_TRIG_8(CLK := EDTTVT1109.status.auto_mode);
	IF R_TRIG_8.Q THEN
		MTBasicsPID_6.Enable := TRUE;
	END_IF;
	F_TRIG_8(CLK := EDTTVT1109.status.auto_mode);
	IF F_TRIG_8.Q THEN
		MTBasicsPID_6.Enable := FALSE;
	END_IF;
	//	MTBasicsPID_6.Enable := TRUE;
	MTBasicsPID_6.Invert := TRUE;
	MTBasicsPID_6.PIDParameters.Gain := EDTPid1109Para.gain;
	MTBasicsPID_6.PIDParameters.IntegrationTime := EDTPid1109Para.integration_time;
	MTBasicsPID_6.PIDParameters.DerivativeTime := EDTPid1109Para.derivative_time;
	MTBasicsPID_6.MinOut := 0.0;
	MTBasicsPID_6.MaxOut := 100.0;
	MTBasicsPID_6.ActValue := EDTTIT1109.status.value;
	MTBasicsPID_6.SetValue := EDTPid1109Para.set_value;
	MTBasicsPID_6.Update := EDTPid1109.update;
	MTBasicsPID_6();
	EDTPid1109.out := MTBasicsPID_6.Out;
	IF MTBasicsPID_6.Active THEN
		EDTTVT1109.input.auto_degree_set := MTBasicsPID_6.Out;
		//	ELSE
		//		EDTTVT1109.input.auto_degree_set := 0.0;
	END_IF;
	IF MTBasicsPID_6.UpdateDone THEN
		EDTPid1109.update := FALSE;
	END_IF;

	//FVT1105 pid调节
	R_TRIG_9(CLK := EDTFVT1105.status.auto_mode);
	IF R_TRIG_9.Q THEN
		MTBasicsPID_12.Enable := TRUE;
	END_IF;
	F_TRIG_9(CLK := EDTFVT1105.status.auto_mode);
	IF F_TRIG_9.Q THEN
		MTBasicsPID_12.Enable := FALSE;
	END_IF;
	//	MTBasicsPID_12.Enable := TRUE;
	MTBasicsPID_12.PIDParameters.Gain := EDTPidFVT1105Para.gain;
	MTBasicsPID_12.PIDParameters.IntegrationTime := EDTPidFVT1105Para.integration_time;
	MTBasicsPID_12.PIDParameters.DerivativeTime := EDTPidFVT1105Para.derivative_time;
	MTBasicsPID_12.MinOut := 0.0;
	MTBasicsPID_12.MaxOut := 100.0;
	MTBasicsPID_12.SetValue := EDTPidFVT1105Para.set_value;
	MTBasicsPID_12.ActValue := EDTFIT1105.flowrate;
	MTBasicsPID_12.Update := EDTPidFVT1105.update;
	MTBasicsPID_12();
	EDTPidFVT1105.out := MTBasicsPID_12.Out;
	IF MTBasicsPID_12.Active THEN
		EDTFVT1105.input.auto_degree_set := MTBasicsPID_12.Out + EDTPidFVT1105Para.min_out;
		//	ELSE
		//		EDTFVT1105.input.auto_degree_set := 0.0;
	END_IF;
	IF MTBasicsPID_12.UpdateDone THEN
		EDTPidFVT1105.update := FALSE;
	END_IF;

	//人工确认步骤可用
	IF (EDTP4S2C.status.run_state) AND (NOT EDTP4S2C_STEP[EDTP4S2C.status.run_step].done AND ((EDTP4S2C.status.run_step = 2) OR (EDTP4S2C.status.run_step = 4) OR (EDTP4S2C.status.run_step = 7)
		OR (EDTP4S2C.status.run_step = 9) OR (EDTP4S2C.status.run_step = 11) OR (p4_step2_5c_confirm_enable))) THEN
		EDTP4S2C.status.confirm_enable := TRUE;
	ELSE
		EDTP4S2C.status.confirm_enable := FALSE;
	END_IF;

END_ACTION
